LIN {X 0,Y 154.831,Z 493.281,A -85,B 0,C 180,E1 -25779.499,E2 -25779.499} C_VEL
LIN {X 0,Y 149.043,Z 503.772,A -85,B 0,C 180,E1 -25782.041,E2 -25782.041} C_VEL
LIN {X 0,Y 142.344,Z 514.195,A -85,B 0,C 180,E1 -25785.287,E2 -25785.287} C_VEL
LIN {X 0,Y 136.226,Z 522.789,A -85,B 0,C 180,E1 -25788.87,E2 -25788.87} C_VEL
LIN {X 0,Y 129.735,Z 531.025,A -85,B 0,C 180,E1 -25793.425,E2 -25793.425} C_VEL
LIN {X 0,Y 124.804,Z 536.98,A -85,B 0,C 180,E1 -25797.884,E2 -25797.884} C_VEL
LIN {X 0,Y 119.794,Z 542.879,A -85,B 0,C 180,E1 -25803.896,E2 -25803.896} C_VEL
LIN {X 0,Y 116.608,Z 546.367,A -85,B 0,C 180,E1 -25808.8,E2 -25808.8} C_VEL
LIN {X 0,Y 113.843,Z 549.761,A -85,B 0,C 180,E1 -25815.704,E2 -25815.704} C_VEL
LIN {X 0,Y 112.436,Z 551.771,A -85,B 0,C 180,E1 -25822.818,E2 -25822.818} C_VEL
LIN {X 0,Y 112.199,Z 552.451,A -85,B 0,C 180,E1 -25830,E2 -25830} C_VEL
LIN {X 0,Y 112.434,Z 551.816,A -85,B 0,C 180,E1 -25837.181,E2 -25837.181} C_VEL
LIN {X 0,Y 113.819,Z 549.846,A -85,B 0,C 180,E1 -25844.299,E2 -25844.299} C_VEL
LIN {X 0,Y 116.58,Z 546.493,A -85,B 0,C 180,E1 -25851.204,E2 -25851.204} C_VEL
LIN {X 0,Y 120.927,Z 541.656,A -85,B 0,C 180,E1 -25857.706,E2 -25857.706} C_VEL
LIN {X 0,Y 126.423,Z 535.183,A -85,B 0,C 180,E1 -25863.773,E2 -25863.773} C_VEL
LIN {X 0,Y 132.35,Z 527.972,A -85,B 0,C 180,E1 -25868.603,E2 -25868.603} C_VEL
LIN {X 0,Y 139.146,Z 519.048,A -85,B 0,C 180,E1 -25872.988,E2 -25872.988} C_VEL
LIN {X 0,Y 145.538,Z 509.671,A -85,B 0,C 180,E1 -25876.413,E2 -25876.413} C_VEL
LIN {X 0,Y 151.745,Z 499.424,A -85,B 0,C 180,E1 -25879.256,E2 -25879.256} C_VEL
LIN {X 0,Y 157.702,Z 487.826,A -85,B 0,C 180,E1 -25881.761,E2 -25881.761} C_VEL
LIN {X 0,Y 163.296,Z 475.115,A -85,B 0,C 180,E1 -25883.799,E2 -25883.799} C_VEL
LIN {X 0,Y 167.805,Z 462.736,A -85,B 0,C 180,E1 -25885.277,E2 -25885.277} C_VEL
LIN {X 0,Y 171.372,Z 450.293,A -85,B 0,C 180,E1 -25886.408,E2 -25886.408} C_VEL
LIN {X 0,Y 174.368,Z 436.456,A -85,B 0,C 180,E1 -25887.284,E2 -25887.284} C_VEL
LIN {X 0,Y 176.327,Z 422.007,A -85,B 0,C 180,E1 -25887.898,E2 -25887.898} C_VEL
LIN {X 0,Y 179.543,Z 385.834,A -85,B 0,C 180,E1 -25888.964,E2 -25888.964} C_VEL
LIN {X 0,Y 177.542,Z 380.775,A -85,B 0,C 180,E1 -25890.461,E2 -25890.461} C_VEL
LIN {X 0,Y 173.513,Z 372.831,A -85,B 0,C 180,E1 -25893.622,E2 -25893.622} C_VEL
LIN {X 0,Y 169.768,Z 366.134,A -85,B 0,C 180,E1 -25897.004,E2 -25897.004} C_VEL
LIN {X 0,Y 166.328,Z 360.29,A -85,B 0,C 180,E1 -25900.724,E2 -25900.724} C_VEL
LIN {X 0,Y 163.415,Z 355.804,A -85,B 0,C 180,E1 -25904.621,E2 -25904.621} C_VEL
LIN {X 0,Y 161.232,Z 352.232,A -85,B 0,C 180,E1 -25908.528,E2 -25908.528} C_VEL
LIN {X 0,Y 158.664,Z 347.179,A -85,B 0,C 180,E1 -25919.365,E2 -25919.365} C_VEL
LIN {X 0,Y 158.668,Z 347.413,A -85,B 0,C 180,E1 -25921.269,E2 -25921.269} C_VEL
LIN {X 0,Y 161.202,Z 352.144,A -85,B 0,C 180,E1 -25931.314,E2 -25931.314} C_VEL
LIN {X 0,Y 163.612,Z 356.049,A -85,B 0,C 180,E1 -25935.581,E2 -25935.581} C_VEL
LIN {X 0,Y 166.843,Z 361.285,A -85,B 0,C 180,E1 -25939.813,E2 -25939.813} C_VEL
LIN {X 0,Y 169.27,Z 365.259,A -85,B 0,C 180,E1 -25942.412,E2 -25942.412} C_VEL
LIN {X 0,Y 172.886,Z 371.75,A -85,B 0,C 180,E1 -25945.767,E2 -25945.767} C_VEL
LIN {X 0,Y 174.889,Z 375.758,A -85,B 0,C 180,E1 -25947.444,E2 -25947.444} C_VEL
LIN {X 0,Y 177.962,Z 383.47,A -85,B 0,C 180,E1 -25949.905,E2 -25949.905} C_VEL
LIN {X 0,Y 179.384,Z 387.559,A -85,B 0,C 180,E1 -25950.996,E2 -25950.996} C_VEL
LIN {X 0,Y 175.579,Z 429.688,A -85,B 0,C 180,E1 -25952.309,E2 -25952.309} C_VEL
LIN {X 0,Y 173.1,Z 443.982,A -85,B 0,C 180,E1 -25953.004,E2 -25953.004} C_VEL
LIN {X 0,Y 169.543,Z 457.949,A -85,B 0,C 180,E1 -25954.001,E2 -25954.001} C_VEL
LIN {X 0,Y 164.994,Z 471.812,A -85,B 0,C 180,E1 -25955.45,E2 -25955.45} C_VEL
LIN {X 0,Y 159.867,Z 484.227,A -85,B 0,C 180,E1 -25957.176,E2 -25957.176} C_VEL
LIN {X 0,Y 154.341,Z 495.58,A -85,B 0,C 180,E1 -25959.278,E2 -25959.278} C_VEL
LIN {X 0,Y 148.493,Z 506.017,A -85,B 0,C 180,E1 -25961.806,E2 -25961.806} C_VEL
LIN {X 0,Y 141.881,Z 516.403,A -85,B 0,C 180,E1 -25965.102,E2 -25965.102} C_VEL
LIN {X 0,Y 135.687,Z 524.971,A -85,B 0,C 180,E1 -25968.671,E2 -25968.671} C_VEL
LIN {X 0,Y 129.237,Z 533.17,A -85,B 0,C 180,E1 -25973.261,E2 -25973.261} C_VEL
LIN {X 0,Y 123.346,Z 540.219,A -85,B 0,C 180,E1 -25978.723,E2 -25978.723} C_VEL
LIN {X 0,Y 119.298,Z 545.014,A -85,B 0,C 180,E1 -25983.78,E2 -25983.78} C_VEL
LIN {X 0,Y 116.235,Z 548.502,A -85,B 0,C 180,E1 -25988.73,E2 -25988.73} C_VEL
LIN {X 0,Y 113.556,Z 551.894,A -85,B 0,C 180,E1 -25995.667,E2 -25995.667} C_VEL
LIN {X 0,Y 112.263,Z 553.898,A -85,B 0,C 180,E1 -26002.808,E2 -26002.808} C_VEL
LIN {X 0,Y 112.133,Z 554.556,A -85,B 0,C 180,E1 -26010,E2 -26010} C_VEL
LIN {X 0,Y 112.278,Z 553.828,A -85,B 0,C 180,E1 -26017.38,E2 -26017.38} C_VEL
LIN {X 0,Y 113.582,Z 551.845,A -85,B 0,C 180,E1 -26024.33,E2 -26024.33} C_VEL
LIN {X 0,Y 116.237,Z 548.428,A -85,B 0,C 180,E1 -26031.271,E2 -26031.271} C_VEL
LIN {X 0,Y 116.783,Z 547.806,A -85,B 0,C 180,E1 -26032.245,E2 -26032.245} C_VEL
LIN {X 0,Y 117.755,Z 546.031,A -85,B 0,C 180,E1 -26034.955,E2 -26034.955} C_VEL
LIN {X 0,Y 118.012,Z 542.788,A -85,B 0,C 180,E1 -26039.51,E2 -26039.51} C_VEL
LIN {X 0,Y 118.831,Z 538.965,A -85,B 0,C 180,E1 -26043.93,E2 -26043.93} C_VEL
LIN {X 0,Y 120.612,Z 536.281,A -85,B 0,C 180,E1 -26046.303,E2 -26046.303} C_VEL
LIN {X 0,Y 126.397,Z 529.621,A -85,B 0,C 180,E1 -26050.792,E2 -26050.792} C_VEL
LIN {X 0,Y 133.529,Z 520.595,A -85,B 0,C 180,E1 -26055.278,E2 -26055.278} C_VEL
LIN {X 0,Y 140.331,Z 511.13,A -85,B 0,C 180,E1 -26058.695,E2 -26058.695} C_VEL
LIN {X 0,Y 146.494,Z 501.341,A -85,B 0,C 180,E1 -26061.416,E2 -26061.416} C_VEL
LIN {X 0,Y 152.443,Z 490.369,A -85,B 0,C 180,E1 -26063.782,E2 -26063.782} C_VEL
LIN {X 0,Y 158.317,Z 477.817,A -85,B 0,C 180,E1 -26065.77,E2 -26065.77} C_VEL
LIN {X 0,Y 162.993,Z 465.66,A -85,B 0,C 180,E1 -26067.224,E2 -26067.224} C_VEL
LIN {X 0,Y 167.084,Z 452.297,A -85,B 0,C 180,E1 -26068.396,E2 -26068.396} C_VEL
LIN {X 0,Y 170.16,Z 438.671,A -85,B 0,C 180,E1 -26069.249,E2 -26069.249} C_VEL
LIN {X 0,Y 172.249,Z 424.594,A -85,B 0,C 180,E1 -26069.814,E2 -26069.814} C_VEL
LIN {X 0,Y 175.377,Z 390.18,A -85,B 0,C 180,E1 -26070.85,E2 -26070.85} C_VEL
LIN {X 0,Y 172.372,Z 381.864,A -85,B 0,C 180,E1 -26073.435,E2 -26073.435} C_VEL
LIN {X 0,Y 170.665,Z 378.041,A -85,B 0,C 180,E1 -26074.969,E2 -26074.969} C_VEL
LIN {X 0,Y 167.157,Z 371.404,A -85,B 0,C 180,E1 -26078.415,E2 -26078.415} C_VEL
LIN {X 0,Y 164.04,Z 366.093,A -85,B 0,C 180,E1 -26082.065,E2 -26082.065} C_VEL
LIN {X 0,Y 161.76,Z 362.326,A -85,B 0,C 180,E1 -26085.373,E2 -26085.373} C_VEL
LIN {X 0,Y 159.691,Z 358.606,A -85,B 0,C 180,E1 -26089.38,E2 -26089.38} C_VEL
LIN {X 0,Y 157.511,Z 354.085,A -85,B 0,C 180,E1 -26098.722,E2 -26098.722} C_VEL
LIN {X 0,Y 157.506,Z 354.034,A -85,B 0,C 180,E1 -26101.279,E2 -26101.279} C_VEL
LIN {X 0,Y 159.956,Z 359.128,A -85,B 0,C 180,E1 -26111.404,E2 -26111.404} C_VEL
LIN {X 0,Y 162.479,Z 363.489,A -85,B 0,C 180,E1 -26115.926,E2 -26115.926} C_VEL
LIN {X 0,Y 164.967,Z 367.653,A -85,B 0,C 180,E1 -26119.279,E2 -26119.279} C_VEL
LIN {X 0,Y 167.552,Z 372.121,A -85,B 0,C 180,E1 -26122.18,E2 -26122.18} C_VEL
LIN {X 0,Y 171.277,Z 379.139,A -85,B 0,C 180,E1 -26125.746,E2 -26125.746} C_VEL
LIN {X 0,Y 175.153,Z 387.363,A -85,B 0,C 180,E1 -26128.962,E2 -26128.962} C_VEL
LIN {X 0,Y 175.509,Z 388.434,A -85,B 0,C 180,E1 -26129.26,E2 -26129.26} C_VEL
LIN {X 0,Y 171.755,Z 428.026,A -85,B 0,C 180,E1 -26130.46,E2 -26130.46} C_VEL
LIN {X 0,Y 169.296,Z 442.095,A -85,B 0,C 180,E1 -26131.155,E2 -26131.155} C_VEL
LIN {X 0,Y 165.594,Z 456.476,A -85,B 0,C 180,E1 -26132.204,E2 -26132.204} C_VEL
LIN {X 0,Y 161.246,Z 469.396,A -85,B 0,C 180,E1 -26133.534,E2 -26133.534} C_VEL
LIN {X 0,Y 156.036,Z 481.927,A -85,B 0,C 180,E1 -26135.279,E2 -26135.279} C_VEL
LIN {X 0,Y 150.311,Z 493.509,A -85,B 0,C 180,E1 -26137.433,E2 -26137.433} C_VEL
LIN {X 0,Y 144.379,Z 503.842,A -85,B 0,C 180,E1 -26139.946,E2 -26139.946} C_VEL
LIN {X 0,Y 137.381,Z 514.264,A -85,B 0,C 180,E1 -26143.199,E2 -26143.199} C_VEL
LIN {X 0,Y 130.954,Z 522.858,A -85,B 0,C 180,E1 -26146.823,E2 -26146.823} C_VEL
LIN {X 0,Y 124.087,Z 531.093,A -85,B 0,C 180,E1 -26151.464,E2 -26151.464} C_VEL
LIN {X 0,Y 119.119,Z 536.642,A -85,B 0,C 180,E1 -26155.691,E2 -26155.691} C_VEL
LIN {X 0,Y 114.718,Z 541.549,A -85,B 0,C 180,E1 -26160.653,E2 -26160.653} C_VEL
LIN {X 0,Y 109.986,Z 546.435,A -85,B 0,C 180,E1 -26167.456,E2 -26167.456} C_VEL
LIN {X 0,Y 106.95,Z 549.829,A -85,B 0,C 180,E1 -26174.761,E2 -26174.761} C_VEL
LIN {X 0,Y 105.378,Z 551.838,A -85,B 0,C 180,E1 -26182.335,E2 -26182.335} C_VEL
LIN {X 0,Y 105.106,Z 552.518,A -85,B 0,C 180,E1 -26190,E2 -26190} C_VEL
LIN {X 0,Y 105.373,Z 551.883,A -85,B 0,C 180,E1 -26197.665,E2 -26197.665} C_VEL
LIN {X 0,Y 106.929,Z 549.912,A -85,B 0,C 180,E1 -26205.242,E2 -26205.242} C_VEL
LIN {X 0,Y 109.96,Z 546.559,A -85,B 0,C 180,E1 -26212.549,E2 -26212.549} C_VEL
LIN {X 0,Y 114.642,Z 541.722,A -85,B 0,C 180,E1 -26219.368,E2 -26219.368} C_VEL
LIN {X 0,Y 120.56,Z 535.248,A -85,B 0,C 180,E1 -26225.657,E2 -26225.657} C_VEL
LIN {X 0,Y 126.86,Z 528.037,A -85,B 0,C 180,E1 -26230.612,E2 -26230.612} C_VEL
LIN {X 0,Y 134.008,Z 519.113,A -85,B 0,C 180,E1 -26235.071,E2 -26235.071} C_VEL
LIN {X 0,Y 140.732,Z 509.734,A -85,B 0,C 180,E1 -26238.509,E2 -26238.509} C_VEL
LIN {X 0,Y 146.984,Z 499.861,A -85,B 0,C 180,E1 -26241.268,E2 -26241.268} C_VEL
LIN {X 0,Y 153.404,Z 487.888,A -85,B 0,C 180,E1 -26243.847,E2 -26243.847} C_VEL
LIN {X 0,Y 159.21,Z 475.176,A -85,B 0,C 180,E1 -26245.859,E2 -26245.859} C_VEL
LIN {X 0,Y 163.865,Z 462.797,A -85,B 0,C 180,E1 -26247.317,E2 -26247.317} C_VEL
LIN {X 0,Y 167.556,Z 450.351,A -85,B 0,C 180,E1 -26248.427,E2 -26248.427} C_VEL
LIN {X 0,Y 170.642,Z 436.511,A -85,B 0,C 180,E1 -26249.286,E2 -26249.286} C_VEL
LIN {X 0,Y 172.672,Z 422.053,A -85,B 0,C 180,E1 -26249.887,E2 -26249.887} C_VEL
LIN {X 0,Y 175.751,Z 388.718,A -85,B 0,C 180,E1 -26250.849,E2 -26250.849} C_VEL
LIN {X 0,Y 173.862,Z 384.198,A -85,B 0,C 180,E1 -26252.38,E2 -26252.38} C_VEL
LIN {X 0,Y 169.806,Z 376.049,A -85,B 0,C 180,E1 -26255.944,E2 -26255.944} C_VEL
LIN {X 0,Y 166.416,Z 369.87,A -85,B 0,C 180,E1 -26259.448,E2 -26259.448} C_VEL
LIN {X 0,Y 164.261,Z 366.273,A -85,B 0,C 180,E1 -26262.058,E2 -26262.058} C_VEL
LIN {X 0,Y 161.985,Z 362.452,A -85,B 0,C 180,E1 -26265.393,E2 -26265.393} C_VEL
LIN {X 0,Y 159.727,Z 358.589,A -85,B 0,C 180,E1 -26269.863,E2 -26269.863} C_VEL
LIN {X 0,Y 157.802,Z 354.129,A -85,B 0,C 180,E1 -26280,E2 -26280} C_VEL
LIN {X 0,Y 160.021,Z 358.971,A -85,B 0,C 180,E1 -26290.718,E2 -26290.718} C_VEL
LIN {X 0,Y 162.659,Z 363.601,A -85,B 0,C 180,E1 -26295.593,E2 -26295.593} C_VEL
LIN {X 0,Y 165.295,Z 368.002,A -85,B 0,C 180,E1 -26299.159,E2 -26299.159} C_VEL
LIN {X 0,Y 168.289,Z 373.184,A -85,B 0,C 180,E1 -26302.471,E2 -26302.471} C_VEL
LIN {X 0,Y 171.793,Z 380.078,A -85,B 0,C 180,E1 -26305.797,E2 -26305.797} C_VEL
LIN {X 0,Y 174.641,Z 387.517,A -85,B 0,C 180,E1 -26308.301,E2 -26308.301} C_VEL
LIN {X 0,Y 175.601,Z 390.329,A -85,B 0,C 180,E1 -26309.109,E2 -26309.109} C_VEL
LIN {X 0,Y 171.889,Z 429.635,A -85,B 0,C 180,E1 -26310.308,E2 -26310.308} C_VEL
LIN {X 0,Y 169.343,Z 443.925,A -85,B 0,C 180,E1 -26310.991,E2 -26310.991} C_VEL
LIN {X 0,Y 165.677,Z 457.89,A -85,B 0,C 180,E1 -26311.965,E2 -26311.965} C_VEL
LIN {X 0,Y 160.969,Z 471.751,A -85,B 0,C 180,E1 -26313.385,E2 -26313.385} C_VEL
LIN {X 0,Y 155.67,Z 484.165,A -85,B 0,C 180,E1 -26315.089,E2 -26315.089} C_VEL
LIN {X 0,Y 149.929,Z 495.517,A -85,B 0,C 180,E1 -26317.168,E2 -26317.168} C_VEL
LIN {X 0,Y 143.85,Z 505.953,A -85,B 0,C 180,E1 -26319.694,E2 -26319.694} C_VEL
LIN {X 0,Y 136.928,Z 516.338,A -85,B 0,C 180,E1 -26322.998,E2 -26322.998} C_VEL
LIN {X 0,Y 130.406,Z 524.906,A -85,B 0,C 180,E1 -26326.598,E2 -26326.598} C_VEL
LIN {X 0,Y 123.579,Z 533.104,A -85,B 0,C 180,E1 -26331.277,E2 -26331.277} C_VEL
LIN {X 0,Y 118.498,Z 538.854,A -85,B 0,C 180,E1 -26335.707,E2 -26335.707} C_VEL
LIN {X 0,Y 114.217,Z 543.56,A -85,B 0,C 180,E1 -26340.512,E2 -26340.512} C_VEL
LIN {X 0,Y 109.632,Z 548.437,A -85,B 0,C 180,E1 -26347.38,E2 -26347.38} C_VEL
LIN {X 0,Y 106.642,Z 551.828,A -85,B 0,C 180,E1 -26354.716,E2 -26354.716} C_VEL
LIN {X 0,Y 105.221,Z 553.832,A -85,B 0,C 180,E1 -26362.324,E2 -26362.324} C_VEL
LIN {X 0,Y 105.033,Z 554.489,A -85,B 0,C 180,E1 -26370,E2 -26370} C_VEL
LIN {X 0,Y 105.222,Z 553.805,A -85,B 0,C 180,E1 -26377.677,E2 -26377.677} C_VEL
LIN {X 0,Y 106.665,Z 551.778,A -85,B 0,C 180,E1 -26385.281,E2 -26385.281} C_VEL
LIN {X 0,Y 109.633,Z 548.36,A -85,B 0,C 180,E1 -26392.62,E2 -26392.62} C_VEL
LIN {X 0,Y 114.167,Z 543.45,A -85,B 0,C 180,E1 -26399.503,E2 -26399.503} C_VEL
LIN {X 0,Y 118.45,Z 538.716,A -85,B 0,C 180,E1 -26404.309,E2 -26404.309} C_VEL
LIN {X 0,Y 120.612,Z 536.281,A -85,B 0,C 180,E1 -26406.303,E2 -26406.303} C_VEL
LIN {X 0,Y 122.566,Z 533.459,A -85,B 0,C 180,E1 -26408.571,E2 -26408.571} C_VEL
LIN {X 0,Y 124.537,Z 528.588,A -85,B 0,C 180,E1 -26412.492,E2 -26412.492} C_VEL
LIN {X 0,Y 126.904,Z 523.234,A -85,B 0,C 180,E1 -26416.137,E2 -26416.137} C_VEL
LIN {X 0,Y 129.353,Z 519.595,A -85,B 0,C 180,E1 -26417.9,E2 -26417.9} C_VEL
LIN {X 0,Y 136.961,Z 509.277,A -85,B 0,C 180,E1 -26421.492,E2 -26421.492} C_VEL
LIN {X 0,Y 143.63,Z 498.759,A -85,B 0,C 180,E1 -26424.256,E2 -26424.256} C_VEL
LIN {X 0,Y 149.688,Z 487.715,A -85,B 0,C 180,E1 -26426.446,E2 -26426.446} C_VEL
LIN {X 0,Y 155.114,Z 476.163,A -85,B 0,C 180,E1 -26428.159,E2 -26428.159} C_VEL
LIN {X 0,Y 160.305,Z 462.603,A -85,B 0,C 180,E1 -26429.668,E2 -26429.668} C_VEL
LIN {X 0,Y 164.387,Z 448.805,A -85,B 0,C 180,E1 -26430.769,E2 -26430.769} C_VEL
LIN {X 0,Y 167.429,Z 434.454,A -85,B 0,C 180,E1 -26431.527,E2 -26431.527} C_VEL
LIN {X 0,Y 169.386,Z 418.688,A -85,B 0,C 180,E1 -26432.07,E2 -26432.07} C_VEL
LIN {X 0,Y 171.756,Z 393.082,A -85,B 0,C 180,E1 -26432.826,E2 -26432.826} C_VEL
LIN {X 0,Y 169.09,Z 385.396,A -85,B 0,C 180,E1 -26435.389,E2 -26435.389} C_VEL
LIN {X 0,Y 165.703,Z 378.484,A -85,B 0,C 180,E1 -26438.87,E2 -26438.87} C_VEL
LIN {X 0,Y 162.588,Z 372.799,A -85,B 0,C 180,E1 -26442.712,E2 -26442.712} C_VEL
LIN {X 0,Y 160.329,Z 368.884,A -85,B 0,C 180,E1 -26446.211,E2 -26446.211} C_VEL
LIN {X 0,Y 158.475,Z 365.407,A -85,B 0,C 180,E1 -26450.105,E2 -26450.105} C_VEL
LIN {X 0,Y 156.641,Z 361.17,A -85,B 0,C 180,E1 -26458.715,E2 -26458.715} C_VEL
LIN {X 0,Y 156.625,Z 360.935,A -85,B 0,C 180,E1 -26460,E2 -26460} C_VEL
LIN {X 0,Y 156.664,Z 361.526,A -85,B 0,C 180,E1 -26462.25,E2 -26462.25} C_VEL
LIN {X 0,Y 158.792,Z 365.998,A -85,B 0,C 180,E1 -26470.842,E2 -26470.842} C_VEL
LIN {X 0,Y 161.048,Z 370.137,A -85,B 0,C 180,E1 -26475.179,E2 -26475.179} C_VEL
LIN {X 0,Y 163.413,Z 374.316,A -85,B 0,C 180,E1 -26478.574,E2 -26478.574} C_VEL
LIN {X 0,Y 166.258,Z 379.525,A -85,B 0,C 180,E1 -26481.913,E2 -26481.913} C_VEL
LIN {X 0,Y 170.019,Z 387.29,A -85,B 0,C 180,E1 -26485.642,E2 -26485.642} C_VEL
LIN {X 0,Y 171.891,Z 391.502,A -85,B 0,C 180,E1 -26487.297,E2 -26487.297} C_VEL
LIN {X 0,Y 168.155,Z 428.91,A -85,B 0,C 180,E1 -26488.416,E2 -26488.416} C_VEL
LIN {X 0,Y 165.533,Z 443.044,A -85,B 0,C 180,E1 -26489.109,E2 -26489.109} C_VEL
LIN {X 0,Y 161.927,Z 456.55,A -85,B 0,C 180,E1 -26490.081,E2 -26490.081} C_VEL
LIN {X 0,Y 157.437,Z 469.468,A -85,B 0,C 180,E1 -26491.381,E2 -26491.381} C_VEL
LIN {X 0,Y 152.04,Z 481.998,A -85,B 0,C 180,E1 -26493.091,E2 -26493.091} C_VEL
LIN {X 0,Y 146.165,Z 493.423,A -85,B 0,C 180,E1 -26495.175,E2 -26495.175} C_VEL
LIN {X 0,Y 139.922,Z 503.912,A -85,B 0,C 180,E1 -26497.714,E2 -26497.714} C_VEL
LIN {X 0,Y 132.615,Z 514.334,A -85,B 0,C 180,E1 -26500.96,E2 -26500.96} C_VEL
LIN {X 0,Y 125.852,Z 522.927,A -85,B 0,C 180,E1 -26504.603,E2 -26504.603} C_VEL
LIN {X 0,Y 118.592,Z 531.162,A -85,B 0,C 180,E1 -26509.317,E2 -26509.317} C_VEL
LIN {X 0,Y 112.947,Z 537.089,A -85,B 0,C 180,E1 -26513.99,E2 -26513.99} C_VEL
LIN {X 0,Y 107.177,Z 543.015,A -85,B 0,C 180,E1 -26520.541,E2 -26520.541} C_VEL
LIN {X 0,Y 103.436,Z 546.502,A -85,B 0,C 180,E1 -26525.942,E2 -26525.942} C_VEL
LIN {X 0,Y 100.098,Z 549.896,A -85,B 0,C 180,E1 -26533.69,E2 -26533.69} C_VEL
LIN {X 0,Y 98.336,Z 551.905,A -85,B 0,C 180,E1 -26541.782,E2 -26541.782} C_VEL
LIN {X 0,Y 98.006,Z 552.585,A -85,B 0,C 180,E1 -26550,E2 -26550} C_VEL
LIN {X 0,Y 98.33,Z 551.949,A -85,B 0,C 180,E1 -26558.218,E2 -26558.218} C_VEL
LIN {X 0,Y 100.079,Z 549.978,A -85,B 0,C 180,E1 -26566.313,E2 -26566.313} C_VEL
LIN {X 0,Y 103.412,Z 546.625,A -85,B 0,C 180,E1 -26574.064,E2 -26574.064} C_VEL
LIN {X 0,Y 108.469,Z 541.788,A -85,B 0,C 180,E1 -26581.22,E2 -26581.22} C_VEL
LIN {X 0,Y 114.826,Z 535.314,A -85,B 0,C 180,E1 -26587.737,E2 -26587.737} C_VEL
LIN {X 0,Y 121.548,Z 528.102,A -85,B 0,C 180,E1 -26592.795,E2 -26592.795} C_VEL
LIN {X 0,Y 129.068,Z 519.177,A -85,B 0,C 180,E1 -26597.314,E2 -26597.314} C_VEL
LIN {X 0,Y 136.124,Z 509.798,A -85,B 0,C 180,E1 -26600.753,E2 -26600.753} C_VEL
LIN {X 0,Y 143.307,Z 498.715,A -85,B 0,C 180,E1 -26603.808,E2 -26603.808} C_VEL
LIN {X 0,Y 149.972,Z 486.66,A -85,B 0,C 180,E1 -26606.282,E2 -26606.282} C_VEL
LIN {X 0,Y 155.337,Z 475.238,A -85,B 0,C 180,E1 -26608.027,E2 -26608.027} C_VEL
LIN {X 0,Y 160.139,Z 462.857,A -85,B 0,C 180,E1 -26609.458,E2 -26609.458} C_VEL
LIN {X 0,Y 164.264,Z 449.283,A -85,B 0,C 180,E1 -26610.617,E2 -26610.617} C_VEL
LIN {X 0,Y 167.359,Z 435.332,A -85,B 0,C 180,E1 -26611.445,E2 -26611.445} C_VEL
LIN {X 0,Y 169.329,Z 421.189,A -85,B 0,C 180,E1 -26611.994,E2 -26611.994} C_VEL
LIN {X 0,Y 172.133,Z 391.736,A -85,B 0,C 180,E1 -26612.82,E2 -26612.82} C_VEL
LIN {X 0,Y 168.615,Z 384.111,A -85,B 0,C 180,E1 -26616.027,E2 -26616.027} C_VEL
LIN {X 0,Y 165.63,Z 378.137,A -85,B 0,C 180,E1 -26619.176,E2 -26619.176} C_VEL
LIN {X 0,Y 162.68,Z 372.786,A -85,B 0,C 180,E1 -26622.884,E2 -26622.884} C_VEL
LIN {X 0,Y 160.554,Z 369.057,A -85,B 0,C 180,E1 -26626.23,E2 -26626.23} C_VEL
LIN {X 0,Y 158.66,Z 365.533,A -85,B 0,C 180,E1 -26630.277,E2 -26630.277} C_VEL
LIN {X 0,Y 156.934,Z 361.2,A -85,B 0,C 180,E1 -26640,E2 -26640} C_VEL
LIN {X 0,Y 158.886,Z 365.886,A -85,B 0,C 180,E1 -26650.191,E2 -26650.191} C_VEL
LIN {X 0,Y 161.185,Z 370.158,A -85,B 0,C 180,E1 -26654.762,E2 -26654.762} C_VEL
LIN {X 0,Y 163.654,Z 374.504,A -85,B 0,C 180,E1 -26658.343,E2 -26658.343} C_VEL
LIN {X 0,Y 166.29,Z 379.356,A -85,B 0,C 180,E1 -26661.47,E2 -26661.47} C_VEL
LIN {X 0,Y 169.511,Z 386.132,A -85,B 0,C 180,E1 -26664.761,E2 -26664.761} C_VEL
LIN {X 0,Y 171.977,Z 393.158,A -85,B 0,C 180,E1 -26667.12,E2 -26667.12} C_VEL
LIN {X 0,Y 168.347,Z 430.051,A -85,B 0,C 180,E1 -26668.242,E2 -26668.242} C_VEL
LIN {X 0,Y 165.723,Z 444.22,A -85,B 0,C 180,E1 -26668.912,E2 -26668.912} C_VEL
LIN {X 0,Y 162.031,Z 457.83,A -85,B 0,C 180,E1 -26669.834,E2 -26669.834} C_VEL
LIN {X 0,Y 157.161,Z 471.689,A -85,B 0,C 180,E1 -26671.216,E2 -26671.216} C_VEL
LIN {X 0,Y 151.698,Z 484.102,A -85,B 0,C 180,E1 -26672.893,E2 -26672.893} C_VEL
LIN {X 0,Y 145.734,Z 495.453,A -85,B 0,C 180,E1 -26674.935,E2 -26674.935} C_VEL
LIN {X 0,Y 139.42,Z 505.89,A -85,B 0,C 180,E1 -26677.447,E2 -26677.447} C_VEL
LIN {X 0,Y 132.167,Z 516.274,A -85,B 0,C 180,E1 -26680.736,E2 -26680.736} C_VEL
LIN {X 0,Y 125.318,Z 524.841,A -85,B 0,C 180,E1 -26684.355,E2 -26684.355} C_VEL
LIN {X 0,Y 118.101,Z 533.039,A -85,B 0,C 180,E1 -26689.113,E2 -26689.113} C_VEL
LIN {X 0,Y 112.653,Z 538.789,A -85,B 0,C 180,E1 -26693.654,E2 -26693.654} C_VEL
LIN {X 0,Y 106.658,Z 544.882,A -85,B 0,C 180,E1 -26700.384,E2 -26700.384} C_VEL
LIN {X 0,Y 103.097,Z 548.371,A -85,B 0,C 180,E1 -26705.858,E2 -26705.858} C_VEL
LIN {X 0,Y 99.769,Z 551.761,A -85,B 0,C 180,E1 -26713.635,E2 -26713.635} C_VEL
LIN {X 0,Y 98.178,Z 553.765,A -85,B 0,C 180,E1 -26721.769,E2 -26721.769} C_VEL
LIN {X 0,Y 97.94,Z 554.423,A -85,B 0,C 180,E1 -26730,E2 -26730} C_VEL
LIN {X 0,Y 98.179,Z 553.738,A -85,B 0,C 180,E1 -26738.231,E2 -26738.231} C_VEL
LIN {X 0,Y 99.787,Z 551.71,A -85,B 0,C 180,E1 -26746.363,E2 -26746.363} C_VEL
LIN {X 0,Y 103.097,Z 548.293,A -85,B 0,C 180,E1 -26754.143,E2 -26754.143} C_VEL
LIN {X 0,Y 107.998,Z 543.382,A -85,B 0,C 180,E1 -26761.372,E2 -26761.372} C_VEL
LIN {X 0,Y 112.625,Z 538.647,A -85,B 0,C 180,E1 -26766.356,E2 -26766.356} C_VEL
LIN {X 0,Y 119.061,Z 531.788,A -85,B 0,C 180,E1 -26771.61,E2 -26771.61} C_VEL
LIN {X 0,Y 126.365,Z 523.274,A -85,B 0,C 180,E1 -26776.303,E2 -26776.303} C_VEL
LIN {X 0,Y 129.353,Z 519.595,A -85,B 0,C 180,E1 -26777.9,E2 -26777.9} C_VEL
LIN {X 0,Y 131.849,Z 515.843,A -85,B 0,C 180,E1 -26779.549,E2 -26779.549} C_VEL
LIN {X 0,Y 134.662,Z 509.463,A -85,B 0,C 180,E1 -26782.587,E2 -26782.587} C_VEL
LIN {X 0,Y 137.474,Z 502.736,A -85,B 0,C 180,E1 -26785.425,E2 -26785.425} C_VEL
LIN {X 0,Y 139.848,Z 498.27,A -85,B 0,C 180,E1 -26786.724,E2 -26786.724} C_VEL
LIN {X 0,Y 145.882,Z 487.644,A -85,B 0,C 180,E1 -26788.772,E2 -26788.772} C_VEL
LIN {X 0,Y 151.492,Z 476.091,A -85,B 0,C 180,E1 -26790.439,E2 -26790.439} C_VEL
LIN {X 0,Y 156.846,Z 462.53,A -85,B 0,C 180,E1 -26791.902,E2 -26791.902} C_VEL
LIN {X 0,Y 160.898,Z 449.259,A -85,B 0,C 180,E1 -26792.936,E2 -26792.936} C_VEL
LIN {X 0,Y 164.048,Z 435.053,A -85,B 0,C 180,E1 -26793.684,E2 -26793.684} C_VEL
LIN {X 0,Y 166.152,Z 418.942,A -85,B 0,C 180,E1 -26794.219,E2 -26794.219} C_VEL
LIN {X 0,Y 168.328,Z 395.923,A -85,B 0,C 180,E1 -26794.905,E2 -26794.905} C_VEL
LIN {X 0,Y 166.227,Z 389.923,A -85,B 0,C 180,E1 -26797.135,E2 -26797.135} C_VEL
LIN {X 0,Y 163.037,Z 383.162,A -85,B 0,C 180,E1 -26800.811,E2 -26800.811} C_VEL
LIN {X 0,Y 160.716,Z 378.768,A -85,B 0,C 180,E1 -26804.017,E2 -26804.017} C_VEL
LIN {X 0,Y 158.846,Z 375.34,A -85,B 0,C 180,E1 -26807.219,E2 -26807.219} C_VEL
LIN {X 0,Y 157.351,Z 372.252,A -85,B 0,C 180,E1 -26810.682,E2 -26810.682} C_VEL
LIN {X 0,Y 155.76,Z 368.083,A -85,B 0,C 180,E1 -26819.354,E2 -26819.354} C_VEL
LIN {X 0,Y 155.768,Z 368.36,A -85,B 0,C 180,E1 -26821.616,E2 -26821.616} C_VEL
LIN {X 0,Y 157.603,Z 372.722,A -85,B 0,C 180,E1 -26830.154,E2 -26830.154} C_VEL
LIN {X 0,Y 159.746,Z 376.961,A -85,B 0,C 180,E1 -26834.589,E2 -26834.589} C_VEL
LIN {X 0,Y 161.937,Z 381.105,A -85,B 0,C 180,E1 -26837.931,E2 -26837.931} C_VEL
LIN {X 0,Y 164.564,Z 386.261,A -85,B 0,C 180,E1 -26841.203,E2 -26841.203} C_VEL
LIN {X 0,Y 167.667,Z 393.111,A -85,B 0,C 180,E1 -26844.503,E2 -26844.503} C_VEL
LIN {X 0,Y 168.423,Z 394.879,A -85,B 0,C 180,E1 -26845.238,E2 -26845.238} C_VEL
LIN {X 0,Y 164.912,Z 428.876,A -85,B 0,C 180,E1 -26846.24,E2 -26846.24} C_VEL
LIN {X 0,Y 162.137,Z 443.368,A -85,B 0,C 180,E1 -26846.93,E2 -26846.93} C_VEL
LIN {X 0,Y 158.127,Z 457.753,A -85,B 0,C 180,E1 -26847.953,E2 -26847.953} C_VEL
LIN {X 0,Y 153.167,Z 471.306,A -85,B 0,C 180,E1 -26849.332,E2 -26849.332} C_VEL
LIN {X 0,Y 147.586,Z 483.494,A -85,B 0,C 180,E1 -26851.003,E2 -26851.003} C_VEL
LIN {X 0,Y 141.29,Z 495.1,A -85,B 0,C 180,E1 -26853.173,E2 -26853.173} C_VEL
LIN {X 0,Y 134.398,Z 505.893,A -85,B 0,C 180,E1 -26855.853,E2 -26855.853} C_VEL
LIN {X 0,Y 126.814,Z 515.936,A -85,B 0,C 180,E1 -26859.117,E2 -26859.117} C_VEL
LIN {X 0,Y 119.831,Z 524.272,A -85,B 0,C 180,E1 -26862.853,E2 -26862.853} C_VEL
LIN {X 0,Y 112.272,Z 532.236,A -85,B 0,C 180,E1 -26867.707,E2 -26867.707} C_VEL
LIN {X 0,Y 105.726,Z 538.643,A -85,B 0,C 180,E1 -26873.255,E2 -26873.255} C_VEL
LIN {X 0,Y 99.588,Z 544.321,A -85,B 0,C 180,E1 -26880.397,E2 -26880.397} C_VEL
LIN {X 0,Y 94.901,Z 548.445,A -85,B 0,C 180,E1 -26888.267,E2 -26888.267} C_VEL
LIN {X 0,Y 92.104,Z 551.136,A -85,B 0,C 180,E1 -26896.767,E2 -26896.767} C_VEL
LIN {X 0,Y 90.892,Z 552.477,A -85,B 0,C 180,E1 -26905.565,E2 -26905.565} C_VEL
LIN {X 0,Y 90.914,Z 552.651,A -85,B 0,C 180,E1 -26910,E2 -26910} C_VEL
LIN {X 0,Y 91.312,Z 552.016,A -85,B 0,C 180,E1 -26918.855,E2 -26918.855} C_VEL
LIN {X 0,Y 93.277,Z 550.044,A -85,B 0,C 180,E1 -26927.54,E2 -26927.54} C_VEL
LIN {X 0,Y 96.952,Z 546.691,A -85,B 0,C 180,E1 -26935.78,E2 -26935.78} C_VEL
LIN {X 0,Y 102.43,Z 541.854,A -85,B 0,C 180,E1 -26943.291,E2 -26943.291} C_VEL
LIN {X 0,Y 107.606,Z 537.018,A -85,B 0,C 180,E1 -26948.568,E2 -26948.568} C_VEL
LIN {X 0,Y 114.284,Z 530.394,A -85,B 0,C 180,E1 -26953.773,E2 -26953.773} C_VEL
LIN {X 0,Y 122.043,Z 521.959,A -85,B 0,C 180,E1 -26958.469,E2 -26958.469} C_VEL
LIN {X 0,Y 129.233,Z 513.154,A -85,B 0,C 180,E1 -26962.048,E2 -26962.048} C_VEL
LIN {X 0,Y 136.88,Z 502.484,A -85,B 0,C 180,E1 -26965.234,E2 -26965.234} C_VEL
LIN {X 0,Y 143.459,Z 491.688,A -85,B 0,C 180,E1 -26967.677,E2 -26967.677} C_VEL
LIN {X 0,Y 149.596,Z 479.871,A -85,B 0,C 180,E1 -26969.681,E2 -26969.681} C_VEL
LIN {X 0,Y 155.225,Z 466.82,A -85,B 0,C 180,E1 -26971.307,E2 -26971.307} C_VEL
LIN {X 0,Y 159.775,Z 453.387,A -85,B 0,C 180,E1 -26972.533,E2 -26972.533} C_VEL
LIN {X 0,Y 163.437,Z 438.744,A -85,B 0,C 180,E1 -26973.446,E2 -26973.446} C_VEL
LIN {X 0,Y 165.719,Z 424.485,A -85,B 0,C 180,E1 -26974.063,E2 -26974.063} C_VEL
LIN {X 0,Y 168.657,Z 395.129,A -85,B 0,C 180,E1 -26974.887,E2 -26974.887} C_VEL
LIN {X 0,Y 165.316,Z 387.521,A -85,B 0,C 180,E1 -26978.352,E2 -26978.352} C_VEL
LIN {X 0,Y 162.448,Z 381.803,A -85,B 0,C 180,E1 -26981.85,E2 -26981.85} C_VEL
LIN {X 0,Y 160.797,Z 378.768,A -85,B 0,C 180,E1 -26984.229,E2 -26984.229} C_VEL
LIN {X 0,Y 159.245,Z 375.763,A -85,B 0,C 180,E1 -26986.927,E2 -26986.927} C_VEL
LIN {X 0,Y 157.603,Z 372.471,A -85,B 0,C 180,E1 -26990.697,E2 -26990.697} C_VEL
LIN {X 0,Y 156.064,Z 368.286,A -85,B 0,C 180,E1 -27000,E2 -27000} C_VEL
LIN {X 0,Y 157.755,Z 372.727,A -85,B 0,C 180,E1 -27009.617,E2 -27009.617} C_VEL
LIN {X 0,Y 159.793,Z 376.8,A -85,B 0,C 180,E1 -27013.999,E2 -27013.999} C_VEL
LIN {X 0,Y 162.098,Z 381.151,A -85,B 0,C 180,E1 -27017.588,E2 -27017.588} C_VEL
LIN {X 0,Y 164.498,Z 385.866,A -85,B 0,C 180,E1 -27020.63,E2 -27020.63} C_VEL
LIN {X 0,Y 167.142,Z 391.792,A -85,B 0,C 180,E1 -27023.544,E2 -27023.544} C_VEL
LIN {X 0,Y 168.577,Z 396.09,A -85,B 0,C 180,E1 -27025.063,E2 -27025.063} C_VEL
LIN {X 0,Y 165.146,Z 429.786,A -85,B 0,C 180,E1 -27026.068,E2 -27026.068} C_VEL
LIN {X 0,Y 162.36,Z 444.36,A -85,B 0,C 180,E1 -27026.729,E2 -27026.729} C_VEL
LIN {X 0,Y 158.273,Z 458.901,A -85,B 0,C 180,E1 -27027.713,E2 -27027.713} C_VEL
LIN {X 0,Y 153.603,Z 471.628,A -85,B 0,C 180,E1 -27028.952,E2 -27028.952} C_VEL
LIN {X 0,Y 147.965,Z 484.04,A -85,B 0,C 180,E1 -27030.585,E2 -27030.585} C_VEL
LIN {X 0,Y 141.775,Z 495.39,A -85,B 0,C 180,E1 -27032.575,E2 -27032.575} C_VEL
LIN {X 0,Y 134.599,Z 506.744,A -85,B 0,C 180,E1 -27035.293,E2 -27035.293} C_VEL
LIN {X 0,Y 127.627,Z 516.21,A -85,B 0,C 180,E1 -27038.309,E2 -27038.309} C_VEL
LIN {X 0,Y 120.423,Z 524.776,A -85,B 0,C 180,E1 -27041.92,E2 -27041.92} C_VEL
LIN {X 0,Y 112.803,Z 532.974,A -85,B 0,C 180,E1 -27046.74,E2 -27046.74} C_VEL
LIN {X 0,Y 106.978,Z 538.723,A -85,B 0,C 180,E1 -27051.385,E2 -27051.385} C_VEL
LIN {X 0,Y 102.027,Z 543.428,A -85,B 0,C 180,E1 -27056.561,E2 -27056.561} C_VEL
LIN {X 0,Y 96.619,Z 548.304,A -85,B 0,C 180,E1 -27064.124,E2 -27064.124} C_VEL
LIN {X 0,Y 92.945,Z 551.695,A -85,B 0,C 180,E1 -27072.395,E2 -27072.395} C_VEL
LIN {X 0,Y 91.137,Z 553.699,A -85,B 0,C 180,E1 -27081.128,E2 -27081.128} C_VEL
LIN {X 0,Y 90.84,Z 554.356,A -85,B 0,C 180,E1 -27090,E2 -27090} C_VEL
LIN {X 0,Y 91.139,Z 553.671,A -85,B 0,C 180,E1 -27098.872,E2 -27098.872} C_VEL
LIN {X 0,Y 92.96,Z 551.643,A -85,B 0,C 180,E1 -27107.602,E2 -27107.602} C_VEL
LIN {X 0,Y 96.617,Z 548.225,A -85,B 0,C 180,E1 -27115.877,E2 -27115.877} C_VEL
LIN {X 0,Y 101.957,Z 543.314,A -85,B 0,C 180,E1 -27123.466,E2 -27123.466} C_VEL
LIN {X 0,Y 106.96,Z 538.579,A -85,B 0,C 180,E1 -27128.624,E2 -27128.624} C_VEL
LIN {X 0,Y 113.818,Z 531.719,A -85,B 0,C 180,E1 -27133.999,E2 -27133.999} C_VEL
LIN {X 0,Y 121.541,Z 523.205,A -85,B 0,C 180,E1 -27138.738,E2 -27138.738} C_VEL
LIN {X 0,Y 128.87,Z 514.322,A -85,B 0,C 180,E1 -27142.256,E2 -27142.256} C_VEL
LIN {X 0,Y 136.507,Z 503.56,A -85,B 0,C 180,E1 -27145.46,E2 -27145.46} C_VEL
LIN {X 0,Y 139.848,Z 498.27,A -85,B 0,C 180,E1 -27146.724,E2 -27146.724} C_VEL
LIN {X 0,Y 142.19,Z 493.721,A -85,B 0,C 180,E1 -27147.933,E2 -27147.933} C_VEL
LIN {X 0,Y 144.893,Z 486.142,A -85,B 0,C 180,E1 -27150.252,E2 -27150.252} C_VEL
LIN {X 0,Y 147.436,Z 478.203,A -85,B 0,C 180,E1 -27152.339,E2 -27152.339} C_VEL
LIN {X 0,Y 149.43,Z 473.097,A -85,B 0,C 180,E1 -27153.176,E2 -27153.176} C_VEL
LIN {X 0,Y 154.384,Z 460.345,A -85,B 0,C 180,E1 -27154.41,E2 -27154.41} C_VEL
LIN {X 0,Y 158.559,Z 446.121,A -85,B 0,C 180,E1 -27155.422,E2 -27155.422} C_VEL
LIN {X 0,Y 161.671,Z 431.162,A -85,B 0,C 180,E1 -27156.076,E2 -27156.076} C_VEL
LIN {X 0,Y 164.201,Z 408.388,A -85,B 0,C 180,E1 -27156.778,E2 -27156.778} C_VEL
LIN {X 0,Y 165.111,Z 398.943,A -85,B 0,C 180,E1 -27157.064,E2 -27157.064} C_VEL
LIN {X 0,Y 163.812,Z 395.201,A -85,B 0,C 180,E1 -27158.592,E2 -27158.592} C_VEL
LIN {X 0,Y 161.056,Z 388.95,A -85,B 0,C 180,E1 -27162.102,E2 -27162.102} C_VEL
LIN {X 0,Y 159.089,Z 385.114,A -85,B 0,C 180,E1 -27165.072,E2 -27165.072} C_VEL
LIN {X 0,Y 157.645,Z 382.166,A -85,B 0,C 180,E1 -27167.775,E2 -27167.775} C_VEL
LIN {X 0,Y 156.239,Z 379.127,A -85,B 0,C 180,E1 -27171.268,E2 -27171.268} C_VEL
LIN {X 0,Y 154.89,Z 375.171,A -85,B 0,C 180,E1 -27179.35,E2 -27179.35} C_VEL
LIN {X 0,Y 154.888,Z 375.364,A -85,B 0,C 180,E1 -27181.3,E2 -27181.3} C_VEL
LIN {X 0,Y 156.525,Z 379.771,A -85,B 0,C 180,E1 -27189.734,E2 -27189.734} C_VEL
LIN {X 0,Y 158.356,Z 383.598,A -85,B 0,C 180,E1 -27193.801,E2 -27193.801} C_VEL
LIN {X 0,Y 160.223,Z 387.359,A -85,B 0,C 180,E1 -27196.894,E2 -27196.894} C_VEL
LIN {X 0,Y 162.526,Z 392.199,A -85,B 0,C 180,E1 -27200.025,E2 -27200.025} C_VEL
LIN {X 0,Y 165.18,Z 398.432,A -85,B 0,C 180,E1 -27203.114,E2 -27203.114} C_VEL
LIN {X 0,Y 161.927,Z 428.835,A -85,B 0,C 180,E1 -27203.988,E2 -27203.988} C_VEL
LIN {X 0,Y 159.11,Z 443.196,A -85,B 0,C 180,E1 -27204.637,E2 -27204.637} C_VEL
LIN {X 0,Y 154.93,Z 457.827,A -85,B 0,C 180,E1 -27205.636,E2 -27205.636} C_VEL
LIN {X 0,Y 149.818,Z 471.378,A -85,B 0,C 180,E1 -27206.966,E2 -27206.966} C_VEL
LIN {X 0,Y 144.063,Z 483.565,A -85,B 0,C 180,E1 -27208.586,E2 -27208.586} C_VEL
LIN {X 0,Y 137.657,Z 494.934,A -85,B 0,C 180,E1 -27210.633,E2 -27210.633} C_VEL
LIN {X 0,Y 130.366,Z 505.963,A -85,B 0,C 180,E1 -27213.323,E2 -27213.323} C_VEL
LIN {X 0,Y 122.45,Z 516.005,A -85,B 0,C 180,E1 -27216.533,E2 -27216.533} C_VEL
LIN {X 0,Y 115.093,Z 524.341,A -85,B 0,C 180,E1 -27220.246,E2 -27220.246} C_VEL
LIN {X 0,Y 107.103,Z 532.305,A -85,B 0,C 180,E1 -27225.139,E2 -27225.139} C_VEL
LIN {X 0,Y 100.085,Z 538.711,A -85,B 0,C 180,E1 -27230.804,E2 -27230.804} C_VEL
LIN {X 0,Y 93.466,Z 544.389,A -85,B 0,C 180,E1 -27238.241,E2 -27238.241} C_VEL
LIN {X 0,Y 88.306,Z 548.513,A -85,B 0,C 180,E1 -27246.551,E2 -27246.551} C_VEL
LIN {X 0,Y 85.201,Z 551.203,A -85,B 0,C 180,E1 -27255.673,E2 -27255.673} C_VEL
LIN {X 0,Y 83.812,Z 552.544,A -85,B 0,C 180,E1 -27265.19,E2 -27265.19} C_VEL
LIN {X 0,Y 83.813,Z 552.718,A -85,B 0,C 180,E1 -27270,E2 -27270} C_VEL
LIN {X 0,Y 84.295,Z 552.082,A -85,B 0,C 180,E1 -27279.598,E2 -27279.598} C_VEL
LIN {X 0,Y 86.494,Z 550.111,A -85,B 0,C 180,E1 -27288.966,E2 -27288.966} C_VEL
LIN {X 0,Y 90.597,Z 546.757,A -85,B 0,C 180,E1 -27297.738,E2 -27297.738} C_VEL
LIN {X 0,Y 96.546,Z 541.919,A -85,B 0,C 180,E1 -27305.615,E2 -27305.615} C_VEL
LIN {X 0,Y 101.759,Z 537.429,A -85,B 0,C 180,E1 -27310.741,E2 -27310.741} C_VEL
LIN {X 0,Y 109.255,Z 530.459,A -85,B 0,C 180,E1 -27316.357,E2 -27316.357} C_VEL
LIN {X 0,Y 117.438,Z 522.023,A -85,B 0,C 180,E1 -27321.073,E2 -27321.073} C_VEL
LIN {X 0,Y 124.994,Z 513.218,A -85,B 0,C 180,E1 -27324.613,E2 -27324.613} C_VEL
LIN {X 0,Y 132.944,Z 502.547,A -85,B 0,C 180,E1 -27327.758,E2 -27327.758} C_VEL
LIN {X 0,Y 139.783,Z 491.751,A -85,B 0,C 180,E1 -27330.143,E2 -27330.143} C_VEL
LIN {X 0,Y 146.146,Z 479.933,A -85,B 0,C 180,E1 -27332.081,E2 -27332.081} C_VEL
LIN {X 0,Y 151.94,Z 466.881,A -85,B 0,C 180,E1 -27333.659,E2 -27333.659} C_VEL
LIN {X 0,Y 156.566,Z 453.676,A -85,B 0,C 180,E1 -27334.816,E2 -27334.816} C_VEL
LIN {X 0,Y 160.321,Z 439.149,A -85,B 0,C 180,E1 -27335.696,E2 -27335.696} C_VEL
LIN {X 0,Y 162.637,Z 425.376,A -85,B 0,C 180,E1 -27336.285,E2 -27336.285} C_VEL
LIN {X 0,Y 165.438,Z 398.675,A -85,B 0,C 180,E1 -27336.997,E2 -27336.997} C_VEL
LIN {X 0,Y 162.296,Z 391.332,A -85,B 0,C 180,E1 -27340.719,E2 -27340.719} C_VEL
LIN {X 0,Y 159.76,Z 386.038,A -85,B 0,C 180,E1 -27344.369,E2 -27344.369} C_VEL
LIN {X 0,Y 157.845,Z 382.269,A -85,B 0,C 180,E1 -27347.872,E2 -27347.872} C_VEL
LIN {X 0,Y 156.363,Z 379.191,A -85,B 0,C 180,E1 -27351.656,E2 -27351.656} C_VEL
LIN {X 0,Y 155.189,Z 375.413,A -85,B 0,C 180,E1 -27360,E2 -27360} C_VEL
LIN {X 0,Y 156.68,Z 379.703,A -85,B 0,C 180,E1 -27369.162,E2 -27369.162} C_VEL
LIN {X 0,Y 158.529,Z 383.676,A -85,B 0,C 180,E1 -27373.418,E2 -27373.418} C_VEL
LIN {X 0,Y 160.45,Z 387.476,A -85,B 0,C 180,E1 -27376.625,E2 -27376.625} C_VEL
LIN {X 0,Y 162.703,Z 392.286,A -85,B 0,C 180,E1 -27379.722,E2 -27379.722} C_VEL
LIN {X 0,Y 164.785,Z 397.347,A -85,B 0,C 180,E1 -27382.225,E2 -27382.225} C_VEL
LIN {X 0,Y 165.409,Z 399.26,A -85,B 0,C 180,E1 -27382.956,E2 -27382.956} C_VEL
LIN {X 0,Y 162.063,Z 430.286,A -85,B 0,C 180,E1 -27383.835,E2 -27383.835} C_VEL
LIN {X 0,Y 159.223,Z 444.596,A -85,B 0,C 180,E1 -27384.466,E2 -27384.466} C_VEL
LIN {X 0,Y 155.088,Z 458.841,A -85,B 0,C 180,E1 -27385.382,E2 -27385.382} C_VEL
LIN {X 0,Y 150.291,Z 471.567,A -85,B 0,C 180,E1 -27386.58,E2 -27386.58} C_VEL
LIN {X 0,Y 144.483,Z 483.978,A -85,B 0,C 180,E1 -27388.162,E2 -27388.162} C_VEL
LIN {X 0,Y 138.08,Z 495.327,A -85,B 0,C 180,E1 -27390.089,E2 -27390.089} C_VEL
LIN {X 0,Y 131.093,Z 505.993,A -85,B 0,C 180,E1 -27392.567,E2 -27392.567} C_VEL
LIN {X 0,Y 123.342,Z 516.145,A -85,B 0,C 180,E1 -27395.714,E2 -27395.714} C_VEL
LIN {X 0,Y 115.778,Z 524.711,A -85,B 0,C 180,E1 -27399.292,E2 -27399.292} C_VEL
LIN {X 0,Y 107.7,Z 532.908,A -85,B 0,C 180,E1 -27404.128,E2 -27404.128} C_VEL
LIN {X 0,Y 101.485,Z 538.657,A -85,B 0,C 180,E1 -27408.862,E2 -27408.862} C_VEL
LIN {X 0,Y 94.512,Z 544.75,A -85,B 0,C 180,E1 -27416.104,E2 -27416.104} C_VEL
LIN {X 0,Y 90.249,Z 548.238,A -85,B 0,C 180,E1 -27422.146,E2 -27422.146} C_VEL
LIN {X 0,Y 86.178,Z 551.628,A -85,B 0,C 180,E1 -27430.962,E2 -27430.962} C_VEL
LIN {X 0,Y 84.123,Z 553.632,A -85,B 0,C 180,E1 -27440.382,E2 -27440.382} C_VEL
LIN {X 0,Y 83.761,Z 554.29,A -85,B 0,C 180,E1 -27450,E2 -27450} C_VEL
LIN {X 0,Y 84.125,Z 553.604,A -85,B 0,C 180,E1 -27459.618,E2 -27459.618} C_VEL
LIN {X 0,Y 86.191,Z 551.575,A -85,B 0,C 180,E1 -27469.036,E2 -27469.036} C_VEL
LIN {X 0,Y 90.245,Z 548.157,A -85,B 0,C 180,E1 -27477.856,E2 -27477.856} C_VEL
LIN {X 0,Y 96.057,Z 543.245,A -85,B 0,C 180,E1 -27485.825,E2 -27485.825} C_VEL
LIN {X 0,Y 103.465,Z 536.698,A -85,B 0,C 180,E1 -27492.785,E2 -27492.785} C_VEL
LIN {X 0,Y 111.073,Z 529.415,A -85,B 0,C 180,E1 -27498.026,E2 -27498.026} C_VEL
LIN {X 0,Y 118.215,Z 521.78,A -85,B 0,C 180,E1 -27501.972,E2 -27501.972} C_VEL
LIN {X 0,Y 125.94,Z 512.624,A -85,B 0,C 180,E1 -27505.396,E2 -27505.396} C_VEL
LIN {X 0,Y 132.602,Z 503.491,A -85,B 0,C 180,E1 -27507.994,E2 -27507.994} C_VEL
LIN {X 0,Y 139.469,Z 492.593,A -85,B 0,C 180,E1 -27510.369,E2 -27510.369} C_VEL
LIN {X 0,Y 145.938,Z 480.66,A -85,B 0,C 180,E1 -27512.236,E2 -27512.236} C_VEL
LIN {X 0,Y 149.43,Z 473.097,A -85,B 0,C 180,E1 -27513.176,E2 -27513.176} C_VEL
LIN {X 0,Y 151.301,Z 467.878,A -85,B 0,C 180,E1 -27513.964,E2 -27513.964} C_VEL
LIN {X 0,Y 153.21,Z 459.317,A -85,B 0,C 180,E1 -27515.72,E2 -27515.72} C_VEL
LIN {X 0,Y 154.803,Z 450.522,A -85,B 0,C 180,E1 -27517.309,E2 -27517.309} C_VEL
LIN {X 0,Y 156.023,Z 444.942,A -85,B 0,C 180,E1 -27517.852,E2 -27517.852} C_VEL
LIN {X 0,Y 158.936,Z 431.021,A -85,B 0,C 180,E1 -27518.418,E2 -27518.418} C_VEL
LIN {X 0,Y 161.656,Z 407.202,A -85,B 0,C 180,E1 -27519.113,E2 -27519.113} C_VEL
LIN {X 0,Y 162.128,Z 402.16,A -85,B 0,C 180,E1 -27519.29,E2 -27519.29} C_VEL
LIN {X 0,Y 159.775,Z 396.242,A -85,B 0,C 180,E1 -27522.48,E2 -27522.48} C_VEL
LIN {X 0,Y 157.678,Z 391.715,A -85,B 0,C 180,E1 -27525.867,E2 -27525.867} C_VEL
LIN {X 0,Y 156.305,Z 388.733,A -85,B 0,C 180,E1 -27528.669,E2 -27528.669} C_VEL
LIN {X 0,Y 155.144,Z 385.994,A -85,B 0,C 180,E1 -27531.862,E2 -27531.862} C_VEL
LIN {X 0,Y 154.025,Z 382.112,A -85,B 0,C 180,E1 -27540,E2 -27540} C_VEL
LIN {X 0,Y 154.153,Z 383.872,A -85,B 0,C 180,E1 -27543.922,E2 -27543.922} C_VEL
LIN {X 0,Y 155.393,Z 386.612,A -85,B 0,C 180,E1 -27549.108,E2 -27549.108} C_VEL
LIN {X 0,Y 157.008,Z 390.26,A -85,B 0,C 180,E1 -27553.023,E2 -27553.023} C_VEL
LIN {X 0,Y 158.803,Z 394.138,A -85,B 0,C 180,E1 -27556.223,E2 -27556.223} C_VEL
LIN {X 0,Y 161.189,Z 399.596,A -85,B 0,C 180,E1 -27559.659,E2 -27559.659} C_VEL
LIN {X 0,Y 162.167,Z 402.047,A -85,B 0,C 180,E1 -27560.909,E2 -27560.909} C_VEL
LIN {X 0,Y 159.169,Z 428.993,A -85,B 0,C 180,E1 -27561.664,E2 -27561.664} C_VEL
LIN {X 0,Y 156.286,Z 443.267,A -85,B 0,C 180,E1 -27562.27,E2 -27562.27} C_VEL
LIN {X 0,Y 152.368,Z 456.772,A -85,B 0,C 180,E1 -27563.132,E2 -27563.132} C_VEL
LIN {X 0,Y 147.489,Z 469.685,A -85,B 0,C 180,E1 -27564.313,E2 -27564.313} C_VEL
LIN {X 0,Y 141.533,Z 482.212,A -85,B 0,C 180,E1 -27565.842,E2 -27565.842} C_VEL
LIN {X 0,Y 135.01,Z 493.634,A -85,B 0,C 180,E1 -27567.758,E2 -27567.758} C_VEL
LIN {X 0,Y 127.996,Z 504.121,A -85,B 0,C 180,E1 -27570.142,E2 -27570.142} C_VEL
LIN {X 0,Y 119.713,Z 514.542,A -85,B 0,C 180,E1 -27573.222,E2 -27573.222} C_VEL
LIN {X 0,Y 111.892,Z 523.134,A -85,B 0,C 180,E1 -27576.791,E2 -27576.791} C_VEL
LIN {X 0,Y 103.324,Z 531.367,A -85,B 0,C 180,E1 -27581.566,E2 -27581.566} C_VEL
LIN {X 0,Y 95.029,Z 538.455,A -85,B 0,C 180,E1 -27587.695,E2 -27587.695} C_VEL
LIN {X 0,Y 89.162,Z 543.219,A -85,B 0,C 180,E1 -27593.76,E2 -27593.76} C_VEL
LIN {X 0,Y 84.391,Z 546.705,A -85,B 0,C 180,E1 -27600.022,E2 -27600.022} C_VEL
LIN {X 0,Y 79.792,Z 550.098,A -85,B 0,C 180,E1 -27609.371,E2 -27609.371} C_VEL
LIN {X 0,Y 77.296,Z 552.106,A -85,B 0,C 180,E1 -27619.523,E2 -27619.523} C_VEL
LIN {X 0,Y 76.735,Z 552.784,A -85,B 0,C 180,E1 -27630,E2 -27630} C_VEL
LIN {X 0,Y 77.29,Z 552.148,A -85,B 0,C 180,E1 -27640.478,E2 -27640.478} C_VEL
LIN {X 0,Y 79.776,Z 550.177,A -85,B 0,C 180,E1 -27650.632,E2 -27650.632} C_VEL
LIN {X 0,Y 84.369,Z 546.823,A -85,B 0,C 180,E1 -27659.986,E2 -27659.986} C_VEL
LIN {X 0,Y 90.845,Z 541.985,A -85,B 0,C 180,E1 -27668.234,E2 -27668.234} C_VEL
LIN {X 0,Y 98.768,Z 535.51,A -85,B 0,C 180,E1 -27675.361,E2 -27675.361} C_VEL
LIN {X 0,Y 106.839,Z 528.297,A -85,B 0,C 180,E1 -27680.616,E2 -27680.616} C_VEL
LIN {X 0,Y 114.367,Z 520.737,A -85,B 0,C 180,E1 -27684.509,E2 -27684.509} C_VEL
LIN {X 0,Y 122.365,Z 511.658,A -85,B 0,C 180,E1 -27687.902,E2 -27687.902} C_VEL
LIN {X 0,Y 130.386,Z 501.045,A -85,B 0,C 180,E1 -27690.837,E2 -27690.837} C_VEL
LIN {X 0,Y 137.818,Z 489.428,A -85,B 0,C 180,E1 -27693.175,E2 -27693.175} C_VEL
LIN {X 0,Y 144.451,Z 477.002,A -85,B 0,C 180,E1 -27694.978,E2 -27694.978} C_VEL
LIN {X 0,Y 149.679,Z 465.023,A -85,B 0,C 180,E1 -27696.287,E2 -27696.287} C_VEL
LIN {X 0,Y 154.219,Z 451.945,A -85,B 0,C 180,E1 -27697.319,E2 -27697.319} C_VEL
LIN {X 0,Y 157.872,Z 437.584,A -85,B 0,C 180,E1 -27698.121,E2 -27698.121} C_VEL
LIN {X 0,Y 160.144,Z 423.754,A -85,B 0,C 180,E1 -27698.643,E2 -27698.643} C_VEL
LIN {X 0,Y 162.42,Z 402.343,A -85,B 0,C 180,E1 -27699.204,E2 -27699.204} C_VEL
LIN {X 0,Y 159.974,Z 396.358,A -85,B 0,C 180,E1 -27702.513,E2 -27702.513} C_VEL
LIN {X 0,Y 157.923,Z 391.92,A -85,B 0,C 180,E1 -27705.851,E2 -27705.851} C_VEL
LIN {X 0,Y 156.49,Z 388.757,A -85,B 0,C 180,E1 -27708.832,E2 -27708.832} C_VEL
LIN {X 0,Y 155.302,Z 386.074,A -85,B 0,C 180,E1 -27712.197,E2 -27712.197} C_VEL
LIN {X 0,Y 154.314,Z 382.534,A -85,B 0,C 180,E1 -27720,E2 -27720} C_VEL
LIN {X 0,Y 155.6,Z 386.608,A -85,B 0,C 180,E1 -27728.645,E2 -27728.645} C_VEL
LIN {X 0,Y 157.247,Z 390.438,A -85,B 0,C 180,E1 -27732.749,E2 -27732.749} C_VEL
LIN {X 0,Y 159.12,Z 394.428,A -85,B 0,C 180,E1 -27736.089,E2 -27736.089} C_VEL
LIN {X 0,Y 161.453,Z 399.899,A -85,B 0,C 180,E1 -27739.467,E2 -27739.467} C_VEL
LIN {X 0,Y 162.417,Z 402.492,A -85,B 0,C 180,E1 -27740.724,E2 -27740.724} C_VEL
LIN {X 0,Y 159.301,Z 430.428,A -85,B 0,C 180,E1 -27741.513,E2 -27741.513} C_VEL
LIN {X 0,Y 156.293,Z 445.043,A -85,B 0,C 180,E1 -27742.128,E2 -27742.128} C_VEL
LIN {X 0,Y 152.183,Z 458.782,A -85,B 0,C 180,E1 -27742.969,E2 -27742.969} C_VEL
LIN {X 0,Y 147.25,Z 471.506,A -85,B 0,C 180,E1 -27744.108,E2 -27744.108} C_VEL
LIN {X 0,Y 141.267,Z 483.916,A -85,B 0,C 180,E1 -27745.619,E2 -27745.619} C_VEL
LIN {X 0,Y 134.646,Z 495.264,A -85,B 0,C 180,E1 -27747.463,E2 -27747.463} C_VEL
LIN {X 0,Y 126.921,Z 506.603,A -85,B 0,C 180,E1 -27750.04,E2 -27750.04} C_VEL
LIN {X 0,Y 119.331,Z 516.081,A -85,B 0,C 180,E1 -27752.941,E2 -27752.941} C_VEL
LIN {X 0,Y 111.401,Z 524.647,A -85,B 0,C 180,E1 -27756.453,E2 -27756.453} C_VEL
LIN {X 0,Y 102.864,Z 532.843,A -85,B 0,C 180,E1 -27761.276,E2 -27761.276} C_VEL
LIN {X 0,Y 96.219,Z 538.592,A -85,B 0,C 180,E1 -27766.062,E2 -27766.062} C_VEL
LIN {X 0,Y 90.418,Z 543.296,A -85,B 0,C 180,E1 -27771.552,E2 -27771.552} C_VEL
LIN {X 0,Y 84.007,Z 548.172,A -85,B 0,C 180,E1 -27779.872,E2 -27779.872} C_VEL
LIN {X 0,Y 79.462,Z 551.562,A -85,B 0,C 180,E1 -27789.282,E2 -27789.282} C_VEL
LIN {X 0,Y 77.111,Z 553.566,A -85,B 0,C 180,E1 -27799.498,E2 -27799.498} C_VEL
LIN {X 0,Y 76.673,Z 554.223,A -85,B 0,C 180,E1 -27810,E2 -27810} C_VEL
LIN {X 0,Y 77.113,Z 553.537,A -85,B 0,C 180,E1 -27820.503,E2 -27820.503} C_VEL
LIN {X 0,Y 79.473,Z 551.508,A -85,B 0,C 180,E1 -27830.716,E2 -27830.716} C_VEL
LIN {X 0,Y 84.002,Z 548.089,A -85,B 0,C 180,E1 -27840.131,E2 -27840.131} C_VEL
LIN {X 0,Y 90.348,Z 543.177,A -85,B 0,C 180,E1 -27848.484,E2 -27848.484} C_VEL
LIN {X 0,Y 96.21,Z 538.442,A -85,B 0,C 180,E1 -27853.943,E2 -27853.943} C_VEL
LIN {X 0,Y 104.038,Z 531.582,A -85,B 0,C 180,E1 -27859.46,E2 -27859.46} C_VEL
LIN {X 0,Y 112.658,Z 523.067,A -85,B 0,C 180,E1 -27864.191,E2 -27864.191} C_VEL
LIN {X 0,Y 120.686,Z 514.184,A -85,B 0,C 180,E1 -27867.605,E2 -27867.605} C_VEL
LIN {X 0,Y 128.969,Z 503.421,A -85,B 0,C 180,E1 -27870.678,E2 -27870.678} C_VEL
LIN {X 0,Y 136.084,Z 492.522,A -85,B 0,C 180,E1 -27872.981,E2 -27872.981} C_VEL
LIN {X 0,Y 142.771,Z 480.589,A -85,B 0,C 180,E1 -27874.757,E2 -27874.757} C_VEL
LIN {X 0,Y 148.785,Z 467.352,A -85,B 0,C 180,E1 -27876.232,E2 -27876.232} C_VEL
LIN {X 0,Y 153.759,Z 453.199,A -85,B 0,C 180,E1 -27877.349,E2 -27877.349} C_VEL
LIN {X 0,Y 156.023,Z 444.942,A -85,B 0,C 180,E1 -27877.852,E2 -27877.852} C_VEL
LIN {X 0,Y 157.129,Z 439.285,A -85,B 0,C 180,E1 -27878.335,E2 -27878.335} C_VEL
LIN {X 0,Y 157.816,Z 430.07,A -85,B 0,C 180,E1 -27879.652,E2 -27879.652} C_VEL
LIN {X 0,Y 158.049,Z 420.761,A -85,B 0,C 180,E1 -27880.914,E2 -27880.914} C_VEL
LIN {X 0,Y 158.433,Z 414.951,A -85,B 0,C 180,E1 -27881.302,E2 -27881.302} C_VEL
LIN {X 0,Y 159.344,Z 405.852,A -85,B 0,C 180,E1 -27881.588,E2 -27881.588} C_VEL
LIN {X 0,Y 157.341,Z 400.73,A -85,B 0,C 180,E1 -27884.753,E2 -27884.753} C_VEL
LIN {X 0,Y 155.354,Z 395.947,A -85,B 0,C 180,E1 -27888.757,E2 -27888.757} C_VEL
LIN {X 0,Y 154.068,Z 392.851,A -85,B 0,C 180,E1 -27892.464,E2 -27892.464} C_VEL
LIN {X 0,Y 153.16,Z 389.155,A -85,B 0,C 180,E1 -27900,E2 -27900} C_VEL
LIN {X 0,Y 154.296,Z 393.462,A -85,B 0,C 180,E1 -27908.513,E2 -27908.513} C_VEL
LIN {X 0,Y 155.75,Z 397.051,A -85,B 0,C 180,E1 -27912.362,E2 -27912.362} C_VEL
LIN {X 0,Y 157.349,Z 400.763,A -85,B 0,C 180,E1 -27915.441,E2 -27915.441} C_VEL
LIN {X 0,Y 159.367,Z 405.861,A -85,B 0,C 180,E1 -27918.614,E2 -27918.614} C_VEL
LIN {X 0,Y 156.526,Z 429.958,A -85,B 0,C 180,E1 -27919.271,E2 -27919.271} C_VEL
LIN {X 0,Y 153.445,Z 444.493,A -85,B 0,C 180,E1 -27919.884,E2 -27919.884} C_VEL
LIN {X 0,Y 149.339,Z 457.974,A -85,B 0,C 180,E1 -27920.721,E2 -27920.721} C_VEL
LIN {X 0,Y 143.942,Z 471.522,A -85,B 0,C 180,E1 -27921.927,E2 -27921.927} C_VEL
LIN {X 0,Y 137.84,Z 483.707,A -85,B 0,C 180,E1 -27923.402,E2 -27923.402} C_VEL
LIN {X 0,Y 130.675,Z 495.54,A -85,B 0,C 180,E1 -27925.359,E2 -27925.359} C_VEL
LIN {X 0,Y 123.139,Z 506.102,A -85,B 0,C 180,E1 -27927.794,E2 -27927.794} C_VEL
LIN {X 0,Y 114.563,Z 516.143,A -85,B 0,C 180,E1 -27930.814,E2 -27930.814} C_VEL
LIN {X 0,Y 106.447,Z 524.479,A -85,B 0,C 180,E1 -27934.383,E2 -27934.383} C_VEL
LIN {X 0,Y 97.517,Z 532.442,A -85,B 0,C 180,E1 -27939.219,E2 -27939.219} C_VEL
LIN {X 0,Y 89.452,Z 538.848,A -85,B 0,C 180,E1 -27945.001,E2 -27945.001} C_VEL
LIN {X 0,Y 81.707,Z 544.525,A -85,B 0,C 180,E1 -27952.98,E2 -27952.98} C_VEL
LIN {X 0,Y 75.422,Z 548.648,A -85,B 0,C 180,E1 -27962.231,E2 -27962.231} C_VEL
LIN {X 0,Y 71.476,Z 551.338,A -85,B 0,C 180,E1 -27972.844,E2 -27972.844} C_VEL
LIN {X 0,Y 69.674,Z 552.677,A -85,B 0,C 180,E1 -27984.211,E2 -27984.211} C_VEL
LIN {X 0,Y 69.647,Z 552.851,A -85,B 0,C 180,E1 -27990,E2 -27990} C_VEL
LIN {X 0,Y 70.317,Z 552.215,A -85,B 0,C 180,E1 -28001.53,E2 -28001.53} C_VEL
LIN {X 0,Y 73.146,Z 550.243,A -85,B 0,C 180,E1 -28012.601,E2 -28012.601} C_VEL
LIN {X 0,Y 78.29,Z 546.889,A -85,B 0,C 180,E1 -28022.588,E2 -28022.588} C_VEL
LIN {X 0,Y 85.362,Z 542.051,A -85,B 0,C 180,E1 -28031.196,E2 -28031.196} C_VEL
LIN {X 0,Y 93.893,Z 535.576,A -85,B 0,C 180,E1 -28038.46,E2 -28038.46} C_VEL
LIN {X 0,Y 102.471,Z 528.362,A -85,B 0,C 180,E1 -28043.693,E2 -28043.693} C_VEL
LIN {X 0,Y 111.737,Z 519.435,A -85,B 0,C 180,E1 -28048.114,E2 -28048.114} C_VEL
LIN {X 0,Y 120.177,Z 510.053,A -85,B 0,C 180,E1 -28051.304,E2 -28051.304} C_VEL
LIN {X 0,Y 128.288,Z 499.387,A -85,B 0,C 180,E1 -28054.006,E2 -28054.006} C_VEL
LIN {X 0,Y 135.509,Z 488.201,A -85,B 0,C 180,E1 -28056.075,E2 -28056.075} C_VEL
LIN {X 0,Y 142.355,Z 475.484,A -85,B 0,C 180,E1 -28057.767,E2 -28057.767} C_VEL
LIN {X 0,Y 147.746,Z 463.098,A -85,B 0,C 180,E1 -28058.987,E2 -28058.987} C_VEL
LIN {X 0,Y 152.346,Z 449.604,A -85,B 0,C 180,E1 -28059.939,E2 -28059.939} C_VEL
LIN {X 0,Y 155.895,Z 435.104,A -85,B 0,C 180,E1 -28060.672,E2 -28060.672} C_VEL
LIN {X 0,Y 158.081,Z 420.806,A -85,B 0,C 180,E1 -28061.121,E2 -28061.121} C_VEL
LIN {X 0,Y 159.647,Z 406.219,A -85,B 0,C 180,E1 -28061.467,E2 -28061.467} C_VEL
LIN {X 0,Y 157.729,Z 401.227,A -85,B 0,C 180,E1 -28064.493,E2 -28064.493} C_VEL
LIN {X 0,Y 156.047,Z 397.351,A -85,B 0,C 180,E1 -28067.709,E2 -28067.709} C_VEL
LIN {X 0,Y 155.189,Z 395.323,A -85,B 0,C 180,E1 -28069.773,E2 -28069.773} C_VEL
LIN {X 0,Y 154.311,Z 393.024,A -85,B 0,C 180,E1 -28072.558,E2 -28072.558} C_VEL
LIN {X 0,Y 153.437,Z 389.682,A -85,B 0,C 180,E1 -28080,E2 -28080} C_VEL
LIN {X 0,Y 154.485,Z 393.381,A -85,B 0,C 180,E1 -28087.953,E2 -28087.953} C_VEL
LIN {X 0,Y 155.923,Z 397.057,A -85,B 0,C 180,E1 -28091.929,E2 -28091.929} C_VEL
LIN {X 0,Y 157.638,Z 401.026,A -85,B 0,C 180,E1 -28095.267,E2 -28095.267} C_VEL
LIN {X 0,Y 159.66,Z 406.219,A -85,B 0,C 180,E1 -28098.46,E2 -28098.46} C_VEL
LIN {X 0,Y 156.781,Z 430.716,A -85,B 0,C 180,E1 -28099.113,E2 -28099.113} C_VEL
LIN {X 0,Y 153.618,Z 445.533,A -85,B 0,C 180,E1 -28099.704,E2 -28099.704} C_VEL
LIN {X 0,Y 149.172,Z 459.852,A -85,B 0,C 180,E1 -28100.552,E2 -28100.552} C_VEL
LIN {X 0,Y 143.735,Z 473.21,A -85,B 0,C 180,E1 -28101.722,E2 -28101.722} C_VEL
LIN {X 0,Y 137.587,Z 485.272,A -85,B 0,C 180,E1 -28103.158,E2 -28103.158} C_VEL
LIN {X 0,Y 130.028,Z 497.451,A -85,B 0,C 180,E1 -28105.134,E2 -28105.134} C_VEL
LIN {X 0,Y 123.009,Z 507.183,A -85,B 0,C 180,E1 -28107.347,E2 -28107.347} C_VEL
LIN {X 0,Y 114.213,Z 517.527,A -85,B 0,C 180,E1 -28110.52,E2 -28110.52} C_VEL
LIN {X 0,Y 105.99,Z 525.838,A -85,B 0,C 180,E1 -28114.021,E2 -28114.021} C_VEL
LIN {X 0,Y 97.072,Z 533.787,A -85,B 0,C 180,E1 -28118.897,E2 -28118.897} C_VEL
LIN {X 0,Y 89.033,Z 540.187,A -85,B 0,C 180,E1 -28124.732,E2 -28124.732} C_VEL
LIN {X 0,Y 81.2,Z 545.862,A -85,B 0,C 180,E1 -28132.71,E2 -28132.71} C_VEL
LIN {X 0,Y 75.042,Z 549.978,A -85,B 0,C 180,E1 -28142.079,E2 -28142.079} C_VEL
LIN {X 0,Y 71.189,Z 552.667,A -85,B 0,C 180,E1 -28152.773,E2 -28152.773} C_VEL
LIN {X 0,Y 69.573,Z 553.995,A -85,B 0,C 180,E1 -28164.203,E2 -28164.203} C_VEL
LIN {X 0,Y 69.574,Z 554.156,A -85,B 0,C 180,E1 -28170,E2 -28170} C_VEL
LIN {X 0,Y 70.111,Z 553.469,A -85,B 0,C 180,E1 -28181.565,E2 -28181.565} C_VEL
LIN {X 0,Y 72.823,Z 551.44,A -85,B 0,C 180,E1 -28192.707,E2 -28192.707} C_VEL
LIN {X 0,Y 77.916,Z 548.021,A -85,B 0,C 180,E1 -28202.765,E2 -28202.765} C_VEL
LIN {X 0,Y 84.851,Z 543.109,A -85,B 0,C 180,E1 -28211.499,E2 -28211.499} C_VEL
LIN {X 0,Y 93.5,Z 536.561,A -85,B 0,C 180,E1 -28218.733,E2 -28218.733} C_VEL
LIN {X 0,Y 102.101,Z 529.278,A -85,B 0,C 180,E1 -28223.977,E2 -28223.977} C_VEL
LIN {X 0,Y 110.031,Z 521.643,A -85,B 0,C 180,E1 -28227.812,E2 -28227.812} C_VEL
LIN {X 0,Y 118.413,Z 512.485,A -85,B 0,C 180,E1 -28231.095,E2 -28231.095} C_VEL
LIN {X 0,Y 125.64,Z 503.351,A -85,B 0,C 180,E1 -28233.507,E2 -28233.507} C_VEL
LIN {X 0,Y 133.01,Z 492.452,A -85,B 0,C 180,E1 -28235.705,E2 -28235.705} C_VEL
LIN {X 0,Y 139.892,Z 480.518,A -85,B 0,C 180,E1 -28237.387,E2 -28237.387} C_VEL
LIN {X 0,Y 146.069,Z 467.279,A -85,B 0,C 180,E1 -28238.779,E2 -28238.779} C_VEL
LIN {X 0,Y 151.064,Z 453.479,A -85,B 0,C 180,E1 -28239.807,E2 -28239.807} C_VEL
LIN {X 0,Y 154.679,Z 440.028,A -85,B 0,C 180,E1 -28240.51,E2 -28240.51} C_VEL
LIN {X 0,Y 157.193,Z 426.017,A -85,B 0,C 180,E1 -28240.992,E2 -28240.992} C_VEL
LIN {X 0,Y 158.433,Z 414.951,A -85,B 0,C 180,E1 -28241.302,E2 -28241.302} C_VEL
LIN {X 0,Y 158.473,Z 412.61,A -85,B 0,C 180,E1 -28241.584,E2 -28241.584} C_VEL
LIN {X 0,Y 158.104,Z 410.223,A -85,B 0,C 180,E1 -28242.333,E2 -28242.333} C_VEL
LIN {X 0,Y 157.2,Z 407.91,A -85,B 0,C 180,E1 -28243.756,E2 -28243.756} C_VEL
LIN {X 0,Y 154.747,Z 404.422,A -85,B 0,C 180,E1 -28247.946,E2 -28247.946} C_VEL
LIN {X 0,Y 153.625,Z 401.526,A -85,B 0,C 180,E1 -28250.869,E2 -28250.869} C_VEL
LIN {X 0,Y 153.01,Z 399.702,A -85,B 0,C 180,E1 -28253.075,E2 -28253.075} C_VEL
LIN {X 0,Y 152.288,Z 396.256,A -85,B 0,C 180,E1 -28260,E2 -28260} C_VEL
LIN {X 0,Y 153.215,Z 400.312,A -85,B 0,C 180,E1 -28267.91,E2 -28267.91} C_VEL
LIN {X 0,Y 154.553,Z 403.92,A -85,B 0,C 180,E1 -28271.779,E2 -28271.779} C_VEL
LIN {X 0,Y 156.034,Z 407.655,A -85,B 0,C 180,E1 -28274.844,E2 -28274.844} C_VEL
LIN {X 0,Y 156.824,Z 409.84,A -85,B 0,C 180,E1 -28276.259,E2 -28276.259} C_VEL
LIN {X 0,Y 154.297,Z 430.262,A -85,B 0,C 180,E1 -28276.798,E2 -28276.798} C_VEL
LIN {X 0,Y 151.053,Z 445.057,A -85,B 0,C 180,E1 -28277.381,E2 -28277.381} C_VEL
LIN {X 0,Y 146.581,Z 459.177,A -85,B 0,C 180,E1 -28278.21,E2 -28278.21} C_VEL
LIN {X 0,Y 141.45,Z 471.594,A -85,B 0,C 180,E1 -28279.265,E2 -28279.265} C_VEL
LIN {X 0,Y 135.176,Z 483.778,A -85,B 0,C 180,E1 -28280.637,E2 -28280.637} C_VEL
LIN {X 0,Y 128.276,Z 494.898,A -85,B 0,C 180,E1 -28282.36,E2 -28282.36} C_VEL
LIN {X 0,Y 121.473,Z 504.261,A -85,B 0,C 180,E1 -28284.326,E2 -28284.326} C_VEL
LIN {X 0,Y 112.567,Z 514.68,A -85,B 0,C 180,E1 -28287.168,E2 -28287.168} C_VEL
LIN {X 0,Y 103.992,Z 523.272,A -85,B 0,C 180,E1 -28290.497,E2 -28290.497} C_VEL
LIN {X 0,Y 94.493,Z 531.504,A -85,B 0,C 180,E1 -28295.102,E2 -28295.102} C_VEL
LIN {X 0,Y 86.914,Z 537.246,A -85,B 0,C 180,E1 -28299.81,E2 -28299.81} C_VEL
LIN {X 0,Y 78.082,Z 543.355,A -85,B 0,C 180,E1 -28307.542,E2 -28307.542} C_VEL
LIN {X 0,Y 72.428,Z 546.84,A -85,B 0,C 180,E1 -28314.395,E2 -28314.395} C_VEL
LIN {X 0,Y 66.641,Z 550.233,A -85,B 0,C 180,E1 -28325.049,E2 -28325.049} C_VEL
LIN {X 0,Y 63.365,Z 552.24,A -85,B 0,C 180,E1 -28337.184,E2 -28337.184} C_VEL
LIN {X 0,Y 62.548,Z 552.917,A -85,B 0,C 180,E1 -28350,E2 -28350} C_VEL
LIN {X 0,Y 63.358,Z 552.281,A -85,B 0,C 180,E1 -28362.817,E2 -28362.817} C_VEL
LIN {X 0,Y 66.627,Z 550.31,A -85,B 0,C 180,E1 -28374.956,E2 -28374.956} C_VEL
LIN {X 0,Y 72.399,Z 546.955,A -85,B 0,C 180,E1 -28385.621,E2 -28385.621} C_VEL
LIN {X 0,Y 80.137,Z 542.117,A -85,B 0,C 180,E1 -28394.554,E2 -28394.554} C_VEL
LIN {X 0,Y 89.318,Z 535.641,A -85,B 0,C 180,E1 -28401.89,E2 -28401.89} C_VEL
LIN {X 0,Y 98.422,Z 528.427,A -85,B 0,C 180,E1 -28407.035,E2 -28407.035} C_VEL
LIN {X 0,Y 108.149,Z 519.5,A -85,B 0,C 180,E1 -28411.315,E2 -28411.315} C_VEL
LIN {X 0,Y 116.926,Z 510.117,A -85,B 0,C 180,E1 -28414.366,E2 -28414.366} C_VEL
LIN {X 0,Y 125.686,Z 498.96,A -85,B 0,C 180,E1 -28417.021,E2 -28417.021} C_VEL
LIN {X 0,Y 133.561,Z 486.973,A -85,B 0,C 180,E1 -28419.065,E2 -28419.065} C_VEL
LIN {X 0,Y 139.824,Z 475.545,A -85,B 0,C 180,E1 -28420.46,E2 -28420.46} C_VEL
LIN {X 0,Y 145.355,Z 463.158,A -85,B 0,C 180,E1 -28421.596,E2 -28421.596} C_VEL
LIN {X 0,Y 149.84,Z 450.387,A -85,B 0,C 180,E1 -28422.441,E2 -28422.441} C_VEL
LIN {X 0,Y 153.499,Z 436.07,A -85,B 0,C 180,E1 -28423.126,E2 -28423.126} C_VEL
LIN {X 0,Y 155.744,Z 422.32,A -85,B 0,C 180,E1 -28423.551,E2 -28423.551} C_VEL
LIN {X 0,Y 157.099,Z 410.054,A -85,B 0,C 180,E1 -28423.853,E2 -28423.853} C_VEL
LIN {X 0,Y 155.275,Z 405.267,A -85,B 0,C 180,E1 -28427.336,E2 -28427.336} C_VEL
LIN {X 0,Y 153.998,Z 402.019,A -85,B 0,C 180,E1 -28430.537,E2 -28430.537} C_VEL
LIN {X 0,Y 153.214,Z 399.83,A -85,B 0,C 180,E1 -28433.332,E2 -28433.332} C_VEL
LIN {X 0,Y 152.56,Z 396.822,A -85,B 0,C 180,E1 -28440,E2 -28440} C_VEL
LIN {X 0,Y 153.424,Z 400.317,A -85,B 0,C 180,E1 -28447.402,E2 -28447.402} C_VEL
LIN {X 0,Y 154.675,Z 403.757,A -85,B 0,C 180,E1 -28451.196,E2 -28451.196} C_VEL
LIN {X 0,Y 156.339,Z 407.954,A -85,B 0,C 180,E1 -28454.698,E2 -28454.698} C_VEL
LIN {X 0,Y 157.089,Z 410.116,A -85,B 0,C 180,E1 -28456.057,E2 -28456.057} C_VEL
LIN {X 0,Y 154.708,Z 430.079,A -85,B 0,C 180,E1 -28456.613,E2 -28456.613} C_VEL
LIN {X 0,Y 151.571,Z 444.754,A -85,B 0,C 180,E1 -28457.151,E2 -28457.151} C_VEL
LIN {X 0,Y 147.222,Z 458.663,A -85,B 0,C 180,E1 -28457.873,E2 -28457.873} C_VEL
LIN {X 0,Y 142.052,Z 471.384,A -85,B 0,C 180,E1 -28458.883,E2 -28458.883} C_VEL
LIN {X 0,Y 135.731,Z 483.792,A -85,B 0,C 180,E1 -28460.204,E2 -28460.204} C_VEL
LIN {X 0,Y 128.713,Z 495.138,A -85,B 0,C 180,E1 -28461.842,E2 -28461.842} C_VEL
LIN {X 0,Y 120.967,Z 505.767,A -85,B 0,C 180,E1 -28463.997,E2 -28463.997} C_VEL
LIN {X 0,Y 112.234,Z 515.953,A -85,B 0,C 180,E1 -28466.836,E2 -28466.836} C_VEL
LIN {X 0,Y 103.564,Z 524.517,A -85,B 0,C 180,E1 -28470.094,E2 -28470.094} C_VEL
LIN {X 0,Y 94.071,Z 532.713,A -85,B 0,C 180,E1 -28474.737,E2 -28474.737} C_VEL
LIN {X 0,Y 86.51,Z 538.461,A -85,B 0,C 180,E1 -28479.488,E2 -28479.488} C_VEL
LIN {X 0,Y 79.69,Z 543.164,A -85,B 0,C 180,E1 -28485.129,E2 -28485.129} C_VEL
LIN {X 0,Y 72.031,Z 548.04,A -85,B 0,C 180,E1 -28494.169,E2 -28494.169} C_VEL
LIN {X 0,Y 66.275,Z 551.429,A -85,B 0,C 180,E1 -28504.903,E2 -28504.903} C_VEL
LIN {X 0,Y 63.149,Z 553.433,A -85,B 0,C 180,E1 -28517.14,E2 -28517.14} C_VEL
LIN {X 0,Y 62.492,Z 554.09,A -85,B 0,C 180,E1 -28530,E2 -28530} C_VEL
LIN {X 0,Y 63.152,Z 553.402,A -85,B 0,C 180,E1 -28542.86,E2 -28542.86} C_VEL
LIN {X 0,Y 66.283,Z 551.372,A -85,B 0,C 180,E1 -28555.095,E2 -28555.095} C_VEL
LIN {X 0,Y 72.022,Z 547.954,A -85,B 0,C 180,E1 -28565.837,E2 -28565.837} C_VEL
LIN {X 0,Y 79.637,Z 543.041,A -85,B 0,C 180,E1 -28574.91,E2 -28574.91} C_VEL
LIN {X 0,Y 88.948,Z 536.493,A -85,B 0,C 180,E1 -28582.196,E2 -28582.196} C_VEL
LIN {X 0,Y 98.076,Z 529.209,A -85,B 0,C 180,E1 -28587.349,E2 -28587.349} C_VEL
LIN {X 0,Y 106.412,Z 521.574,A -85,B 0,C 180,E1 -28591.055,E2 -28591.055} C_VEL
LIN {X 0,Y 115.135,Z 512.416,A -85,B 0,C 180,E1 -28594.203,E2 -28594.203} C_VEL
LIN {X 0,Y 122.623,Z 503.281,A -85,B 0,C 180,E1 -28596.492,E2 -28596.492} C_VEL
LIN {X 0,Y 130.246,Z 492.382,A -85,B 0,C 180,E1 -28598.558,E2 -28598.558} C_VEL
LIN {X 0,Y 137.316,Z 480.447,A -85,B 0,C 180,E1 -28600.125,E2 -28600.125} C_VEL
LIN {X 0,Y 143.65,Z 467.207,A -85,B 0,C 180,E1 -28601.422,E2 -28601.422} C_VEL
LIN {X 0,Y 148.652,Z 453.77,A -85,B 0,C 180,E1 -28602.351,E2 -28602.351} C_VEL
LIN {X 0,Y 152.445,Z 440.016,A -85,B 0,C 180,E1 -28603.02,E2 -28603.02} C_VEL
LIN {X 0,Y 155.075,Z 425.583,A -85,B 0,C 180,E1 -28603.479,E2 -28603.479} C_VEL
LIN {X 0,Y 156.799,Z 409.83,A -85,B 0,C 180,E1 -28603.951,E2 -28603.951} C_VEL
LIN {X 0,Y 155.155,Z 405.338,A -85,B 0,C 180,E1 -28607.079,E2 -28607.079} C_VEL
LIN {X 0,Y 154.747,Z 404.422,A -85,B 0,C 180,E1 -28607.946,E2 -28607.946} C_VEL
LIN {X 0,Y 154.1,Z 403.49,A -85,B 0,C 180,E1 -28609.346,E2 -28609.346} C_VEL
LIN {X 0,Y 153.151,Z 403.125,A -85,B 0,C 180,E1 -28611.527,E2 -28611.527} C_VEL
LIN {X 0,Y 151.584,Z 404.067,A -85,B 0,C 180,E1 -28616.761,E2 -28616.761} C_VEL
LIN {X 0,Y 151.384,Z 403.832,A -85,B 0,C 180,E1 -28619.026,E2 -28619.026} C_VEL
LIN {X 0,Y 151.4,Z 403.506,A -85,B 0,C 180,E1 -28619.773,E2 -28619.773} C_VEL
LIN {X 0,Y 151.372,Z 404.158,A -85,B 0,C 180,E1 -28621.621,E2 -28621.621} C_VEL
LIN {X 0,Y 152.16,Z 407.21,A -85,B 0,C 180,E1 -28627.339,E2 -28627.339} C_VEL
LIN {X 0,Y 153.179,Z 410.263,A -85,B 0,C 180,E1 -28630.682,E2 -28630.682} C_VEL
LIN {X 0,Y 154.531,Z 414.066,A -85,B 0,C 180,E1 -28633.841,E2 -28633.841} C_VEL
LIN {X 0,Y 152.158,Z 431.712,A -85,B 0,C 180,E1 -28634.293,E2 -28634.293} C_VEL
LIN {X 0,Y 148.86,Z 445.97,A -85,B 0,C 180,E1 -28634.811,E2 -28634.811} C_VEL
LIN {X 0,Y 144.523,Z 459.251,A -85,B 0,C 180,E1 -28635.54,E2 -28635.54} C_VEL
LIN {X 0,Y 139.273,Z 471.667,A -85,B 0,C 180,E1 -28636.512,E2 -28636.512} C_VEL
LIN {X 0,Y 132.836,Z 483.849,A -85,B 0,C 180,E1 -28637.765,E2 -28637.765} C_VEL
LIN {X 0,Y 125.134,Z 495.846,A -85,B 0,C 180,E1 -28639.509,E2 -28639.509} C_VEL
LIN {X 0,Y 117.186,Z 506.241,A -85,B 0,C 180,E1 -28641.633,E2 -28641.633} C_VEL
LIN {X 0,Y 107.979,Z 516.281,A -85,B 0,C 180,E1 -28644.329,E2 -28644.329} C_VEL
LIN {X 0,Y 99.111,Z 524.616,A -85,B 0,C 180,E1 -28647.581,E2 -28647.581} C_VEL
LIN {X 0,Y 89.201,Z 532.578,A -85,B 0,C 180,E1 -28652.117,E2 -28652.117} C_VEL
LIN {X 0,Y 80.001,Z 538.984,A -85,B 0,C 180,E1 -28657.756,E2 -28657.756} C_VEL
LIN {X 0,Y 70.816,Z 544.661,A -85,B 0,C 180,E1 -28665.997,E2 -28665.997} C_VEL
LIN {X 0,Y 63.151,Z 548.784,A -85,B 0,C 180,E1 -28676.19,E2 -28676.19} C_VEL
LIN {X 0,Y 58.014,Z 551.472,A -85,B 0,C 180,E1 -28688.689,E2 -28688.689} C_VEL
LIN {X 0,Y 55.564,Z 552.811,A -85,B 0,C 180,E1 -28702.733,E2 -28702.733} C_VEL
LIN {X 0,Y 55.466,Z 552.984,A -85,B 0,C 180,E1 -28710,E2 -28710} C_VEL
LIN {X 0,Y 56.452,Z 552.347,A -85,B 0,C 180,E1 -28724.417,E2 -28724.417} C_VEL
LIN {X 0,Y 60.25,Z 550.376,A -85,B 0,C 180,E1 -28737.812,E2 -28737.812} C_VEL
LIN {X 0,Y 66.724,Z 547.021,A -85,B 0,C 180,E1 -28749.195,E2 -28749.195} C_VEL
LIN {X 0,Y 75.223,Z 542.182,A -85,B 0,C 180,E1 -28758.366,E2 -28758.366} C_VEL
LIN {X 0,Y 85.108,Z 535.707,A -85,B 0,C 180,E1 -28765.664,E2 -28765.664} C_VEL
LIN {X 0,Y 94.736,Z 528.492,A -85,B 0,C 180,E1 -28770.651,E2 -28770.651} C_VEL
LIN {X 0,Y 104.911,Z 519.564,A -85,B 0,C 180,E1 -28774.734,E2 -28774.734} C_VEL
LIN {X 0,Y 114.027,Z 510.181,A -85,B 0,C 180,E1 -28777.591,E2 -28777.591} C_VEL
LIN {X 0,Y 122.994,Z 499.152,A -85,B 0,C 180,E1 -28780.042,E2 -28780.042} C_VEL
LIN {X 0,Y 131.185,Z 487.036,A -85,B 0,C 180,E1 -28781.971,E2 -28781.971} C_VEL
LIN {X 0,Y 137.615,Z 475.607,A -85,B 0,C 180,E1 -28783.243,E2 -28783.243} C_VEL
LIN {X 0,Y 143.276,Z 463.218,A -85,B 0,C 180,E1 -28784.285,E2 -28784.285} C_VEL
LIN {X 0,Y 148.089,Z 449.688,A -85,B 0,C 180,E1 -28785.106,E2 -28785.106} C_VEL
LIN {X 0,Y 151.772,Z 435.318,A -85,B 0,C 180,E1 -28785.722,E2 -28785.722} C_VEL
LIN {X 0,Y 154.111,Z 420.624,A -85,B 0,C 180,E1 -28786.118,E2 -28786.118} C_VEL
LIN {X 0,Y 154.812,Z 414.247,A -85,B 0,C 180,E1 -28786.276,E2 -28786.276} C_VEL
LIN {X 0,Y 153.275,Z 409.944,A -85,B 0,C 180,E1 -28789.962,E2 -28789.962} C_VEL
LIN {X 0,Y 152.168,Z 406.63,A -85,B 0,C 180,E1 -28794.035,E2 -28794.035} C_VEL
LIN {X 0,Y 151.683,Z 403.961,A -85,B 0,C 180,E1 -28800,E2 -28800} C_VEL
LIN {X 0,Y 152.363,Z 407.126,A -85,B 0,C 180,E1 -28806.746,E2 -28806.746} C_VEL
LIN {X 0,Y 153.432,Z 410.448,A -85,B 0,C 180,E1 -28810.407,E2 -28810.407} C_VEL
LIN {X 0,Y 154.796,Z 414.259,A -85,B 0,C 180,E1 -28813.615,E2 -28813.615} C_VEL
LIN {X 0,Y 154.291,Z 419.276,A -85,B 0,C 180,E1 -28813.81,E2 -28813.81} C_VEL
LIN {X 0,Y 152.041,Z 434.431,A -85,B 0,C 180,E1 -28814.19,E2 -28814.19} C_VEL
LIN {X 0,Y 148.547,Z 448.679,A -85,B 0,C 180,E1 -28814.73,E2 -28814.73} C_VEL
LIN {X 0,Y 143.986,Z 461.886,A -85,B 0,C 180,E1 -28815.425,E2 -28815.425} C_VEL
LIN {X 0,Y 138.299,Z 474.709,A -85,B 0,C 180,E1 -28816.432,E2 -28816.432} C_VEL
LIN {X 0,Y 131.832,Z 486.453,A -85,B 0,C 180,E1 -28817.656,E2 -28817.656} C_VEL
LIN {X 0,Y 124.65,Z 497.325,A -85,B 0,C 180,E1 -28819.2,E2 -28819.2} C_VEL
LIN {X 0,Y 116.057,Z 508.32,A -85,B 0,C 180,E1 -28821.456,E2 -28821.456} C_VEL
LIN {X 0,Y 107.676,Z 517.398,A -85,B 0,C 180,E1 -28823.971,E2 -28823.971} C_VEL
LIN {X 0,Y 98.728,Z 525.709,A -85,B 0,C 180,E1 -28827.153,E2 -28827.153} C_VEL
LIN {X 0,Y 88.81,Z 533.656,A -85,B 0,C 180,E1 -28831.714,E2 -28831.714} C_VEL
LIN {X 0,Y 79.611,Z 540.056,A -85,B 0,C 180,E1 -28837.393,E2 -28837.393} C_VEL
LIN {X 0,Y 70.382,Z 545.731,A -85,B 0,C 180,E1 -28845.656,E2 -28845.656} C_VEL
LIN {X 0,Y 62.806,Z 549.846,A -85,B 0,C 180,E1 -28855.98,E2 -28855.98} C_VEL
LIN {X 0,Y 57.712,Z 552.534,A -85,B 0,C 180,E1 -28868.573,E2 -28868.573} C_VEL
LIN {X 0,Y 55.46,Z 553.862,A -85,B 0,C 180,E1 -28882.72,E2 -28882.72} C_VEL
LIN {X 0,Y 55.393,Z 554.023,A -85,B 0,C 180,E1 -28890,E2 -28890} C_VEL
LIN {X 0,Y 56.243,Z 553.335,A -85,B 0,C 180,E1 -28904.473,E2 -28904.473} C_VEL
LIN {X 0,Y 59.885,Z 551.305,A -85,B 0,C 180,E1 -28917.997,E2 -28917.997} C_VEL
LIN {X 0,Y 66.354,Z 547.886,A -85,B 0,C 180,E1 -28929.456,E2 -28929.456} C_VEL
LIN {X 0,Y 74.828,Z 542.907,A -85,B 0,C 180,E1 -28938.894,E2 -28938.894} C_VEL
LIN {X 0,Y 84.765,Z 536.425,A -85,B 0,C 180,E1 -28946.007,E2 -28946.007} C_VEL
LIN {X 0,Y 94.404,Z 529.14,A -85,B 0,C 180,E1 -28951.012,E2 -28951.012} C_VEL
LIN {X 0,Y 103.155,Z 521.505,A -85,B 0,C 180,E1 -28954.517,E2 -28954.517} C_VEL
LIN {X 0,Y 112.221,Z 512.346,A -85,B 0,C 180,E1 -28957.476,E2 -28957.476} C_VEL
LIN {X 0,Y 121.515,Z 501.227,A -85,B 0,C 180,E1 -28960.022,E2 -28960.022} C_VEL
LIN {X 0,Y 129.423,Z 489.874,A -85,B 0,C 180,E1 -28961.856,E2 -28961.856} C_VEL
LIN {X 0,Y 136.678,Z 477.316,A -85,B 0,C 180,E1 -28963.273,E2 -28963.273} C_VEL
LIN {X 0,Y 142.356,Z 465.15,A -85,B 0,C 180,E1 -28964.298,E2 -28964.298} C_VEL
LIN {X 0,Y 147.428,Z 451.22,A -85,B 0,C 180,E1 -28965.13,E2 -28965.13} C_VEL
LIN {X 0,Y 151.183,Z 436.997,A -85,B 0,C 180,E1 -28965.711,E2 -28965.711} C_VEL
LIN {X 0,Y 153.595,Z 422.654,A -85,B 0,C 180,E1 -28966.086,E2 -28966.086} C_VEL
LIN {X 0,Y 154.521,Z 413.996,A -85,B 0,C 180,E1 -28966.365,E2 -28966.365} C_VEL
LIN {X 0,Y 152.872,Z 409.23,A -85,B 0,C 180,E1 -28970.407,E2 -28970.407} C_VEL
LIN {X 0,Y 151.933,Z 406.452,A -85,B 0,C 180,E1 -28973.86,E2 -28973.86} C_VEL
LIN {X 0,Y 151.4,Z 403.506,A -85,B 0,C 180,E1 -28979.773,E2 -28979.773} C_VEL
LIN {X 0,Y 151.437,Z 403.425,A -85,B 0,C 180,E1 -28981.216,E2 -28981.216} C_VEL
LIN {X 0,Y 151.432,Z 404.789,A -85,B 0,C 180,E1 -28982.972,E2 -28982.972} C_VEL
LIN {X 0,Y 151.42,Z 408.304,A -85,B 0,C 180,E1 -28985.238,E2 -28985.238} C_VEL
LIN {X 0,Y 151.777,Z 415.768,A -85,B 0,C 180,E1 -28989.129,E2 -28989.129} C_VEL
LIN {X 0,Y 152.186,Z 417.649,A -85,B 0,C 180,E1 -28990.54,E2 -28990.54} C_VEL
LIN {X 0,Y 152.476,Z 418.483,A -85,B 0,C 180,E1 -28991.314,E2 -28991.314} C_VEL
LIN {X 0,Y 150.331,Z 433.086,A -85,B 0,C 180,E1 -28991.717,E2 -28991.717} C_VEL
LIN {X 0,Y 147.077,Z 446.508,A -85,B 0,C 180,E1 -28992.152,E2 -28992.152} C_VEL
LIN {X 0,Y 142.378,Z 460.436,A -85,B 0,C 180,E1 -28992.871,E2 -28992.871} C_VEL
LIN {X 0,Y 136.592,Z 473.428,A -85,B 0,C 180,E1 -28993.798,E2 -28993.798} C_VEL
LIN {X 0,Y 129.211,Z 486.557,A -85,B 0,C 180,E1 -28995.108,E2 -28995.108} C_VEL
LIN {X 0,Y 121.273,Z 498.136,A -85,B 0,C 180,E1 -28996.755,E2 -28996.755} C_VEL
LIN {X 0,Y 113.17,Z 508.089,A -85,B 0,C 180,E1 -28998.733,E2 -28998.733} C_VEL
LIN {X 0,Y 103.68,Z 517.833,A -85,B 0,C 180,E1 -29001.245,E2 -29001.245} C_VEL
LIN {X 0,Y 94.507,Z 525.914,A -85,B 0,C 180,E1 -29004.362,E2 -29004.362} C_VEL
LIN {X 0,Y 84.187,Z 533.652,A -85,B 0,C 180,E1 -29008.773,E2 -29008.773} C_VEL
LIN {X 0,Y 73.995,Z 540.172,A -85,B 0,C 180,E1 -29014.742,E2 -29014.742} C_VEL
LIN {X 0,Y 65.858,Z 544.729,A -85,B 0,C 180,E1 -29021.67,E2 -29021.67} C_VEL
LIN {X 0,Y 57.362,Z 548.851,A -85,B 0,C 180,E1 -29032.223,E2 -29032.223} C_VEL
LIN {X 0,Y 51.443,Z 551.539,A -85,B 0,C 180,E1 -29045.805,E2 -29045.805} C_VEL
LIN {X 0,Y 48.525,Z 552.878,A -85,B 0,C 180,E1 -29061.672,E2 -29061.672} C_VEL
LIN {X 0,Y 48.368,Z 553.05,A -85,B 0,C 180,E1 -29069.999,E2 -29069.999} C_VEL
LIN {X 0,Y 49.587,Z 552.414,A -85,B 0,C 180,E1 -29086.466,E2 -29086.466} C_VEL
LIN {X 0,Y 54.044,Z 550.442,A -85,B 0,C 180,E1 -29101.342,E2 -29101.342} C_VEL
LIN {X 0,Y 61.362,Z 547.087,A -85,B 0,C 180,E1 -29113.407,E2 -29113.407} C_VEL
LIN {X 0,Y 70.689,Z 542.248,A -85,B 0,C 180,E1 -29122.688,E2 -29122.688} C_VEL
LIN {X 0,Y 81.302,Z 535.772,A -85,B 0,C 180,E1 -29129.815,E2 -29129.815} C_VEL
LIN {X 0,Y 91.451,Z 528.557,A -85,B 0,C 180,E1 -29134.549,E2 -29134.549} C_VEL
LIN {X 0,Y 102.077,Z 519.629,A -85,B 0,C 180,E1 -29138.349,E2 -29138.349} C_VEL
LIN {X 0,Y 111.509,Z 510.245,A -85,B 0,C 180,E1 -29140.973,E2 -29140.973} C_VEL
LIN {X 0,Y 120.746,Z 499.215,A -85,B 0,C 180,E1 -29143.224,E2 -29143.224} C_VEL
LIN {X 0,Y 129.165,Z 487.098,A -85,B 0,C 180,E1 -29144.965,E2 -29144.965} C_VEL
LIN {X 0,Y 135.738,Z 475.668,A -85,B 0,C 180,E1 -29146.114,E2 -29146.114} C_VEL
LIN {X 0,Y 141.516,Z 463.278,A -85,B 0,C 180,E1 -29147.058,E2 -29147.058} C_VEL
LIN {X 0,Y 146.526,Z 449.433,A -85,B 0,C 180,E1 -29147.805,E2 -29147.805} C_VEL
LIN {X 0,Y 150.271,Z 434.961,A -85,B 0,C 180,E1 -29148.365,E2 -29148.365} C_VEL
LIN {X 0,Y 152.657,Z 419.872,A -85,B 0,C 180,E1 -29148.718,E2 -29148.718} C_VEL
LIN {X 0,Y 152.738,Z 418.647,A -85,B 0,C 180,E1 -29148.856,E2 -29148.856} C_VEL
LIN {X 0,Y 151.726,Z 415.476,A -85,B 0,C 180,E1 -29152.012,E2 -29152.012} C_VEL
LIN {X 0,Y 151.16,Z 413.471,A -85,B 0,C 180,E1 -29154.664,E2 -29154.664} C_VEL
LIN {X 0,Y 150.809,Z 411.085,A -85,B 0,C 180,E1 -29160,E2 -29160} C_VEL
LIN {X 0,Y 151.338,Z 414.005,A -85,B 0,C 180,E1 -29166.165,E2 -29166.165} C_VEL
LIN {X 0,Y 152.226,Z 417.143,A -85,B 0,C 180,E1 -29169.623,E2 -29169.623} C_VEL
LIN {X 0,Y 152.787,Z 418.784,A -85,B 0,C 180,E1 -29171.184,E2 -29171.184} C_VEL
LIN {X 0,Y 150.462,Z 434.383,A -85,B 0,C 180,E1 -29171.575,E2 -29171.575} C_VEL
LIN {X 0,Y 147.36,Z 447.004,A -85,B 0,C 180,E1 -29171.982,E2 -29171.982} C_VEL
LIN {X 0,Y 142.674,Z 460.798,A -85,B 0,C 180,E1 -29172.6,E2 -29172.6} C_VEL
LIN {X 0,Y 137.284,Z 473.027,A -85,B 0,C 180,E1 -29173.433,E2 -29173.433} C_VEL
LIN {X 0,Y 130.679,Z 485.085,A -85,B 0,C 180,E1 -29174.528,E2 -29174.528} C_VEL
LIN {X 0,Y 122.497,Z 497.261,A -85,B 0,C 180,E1 -29176.06,E2 -29176.06} C_VEL
LIN {X 0,Y 114.783,Z 506.979,A -85,B 0,C 180,E1 -29177.827,E2 -29177.827} C_VEL
LIN {X 0,Y 104.983,Z 517.333,A -85,B 0,C 180,E1 -29180.414,E2 -29180.414} C_VEL
LIN {X 0,Y 95.677,Z 525.644,A -85,B 0,C 180,E1 -29183.341,E2 -29183.341} C_VEL
LIN {X 0,Y 85.278,Z 533.591,A -85,B 0,C 180,E1 -29187.636,E2 -29187.636} C_VEL
LIN {X 0,Y 75.486,Z 539.99,A -85,B 0,C 180,E1 -29193.081,E2 -29193.081} C_VEL
LIN {X 0,Y 65.468,Z 545.665,A -85,B 0,C 180,E1 -29201.286,E2 -29201.286} C_VEL
LIN {X 0,Y 57.045,Z 549.78,A -85,B 0,C 180,E1 -29211.977,E2 -29211.977} C_VEL
LIN {X 0,Y 51.125,Z 552.468,A -85,B 0,C 180,E1 -29225.645,E2 -29225.645} C_VEL
LIN {X 0,Y 48.412,Z 553.795,A -85,B 0,C 180,E1 -29241.654,E2 -29241.654} C_VEL
LIN {X 0,Y 48.309,Z 553.957,A -85,B 0,C 180,E1 -29250.001,E2 -29250.001} C_VEL
LIN {X 0,Y 49.367,Z 553.268,A -85,B 0,C 180,E1 -29266.542,E2 -29266.542} C_VEL
LIN {X 0,Y 53.68,Z 551.237,A -85,B 0,C 180,E1 -29281.58,E2 -29281.58} C_VEL
LIN {X 0,Y 60.991,Z 547.818,A -85,B 0,C 180,E1 -29293.739,E2 -29293.739} C_VEL
LIN {X 0,Y 70.229,Z 542.904,A -85,B 0,C 180,E1 -29303.184,E2 -29303.184} C_VEL
LIN {X 0,Y 80.982,Z 536.356,A -85,B 0,C 180,E1 -29310.207,E2 -29310.207} C_VEL
LIN {X 0,Y 91.155,Z 529.071,A -85,B 0,C 180,E1 -29314.945,E2 -29314.945} C_VEL
LIN {X 0,Y 101.847,Z 520.043,A -85,B 0,C 180,E1 -29318.679,E2 -29318.679} C_VEL
LIN {X 0,Y 111.293,Z 510.574,A -85,B 0,C 180,E1 -29321.3,E2 -29321.3} C_VEL
LIN {X 0,Y 120.065,Z 500.087,A -85,B 0,C 180,E1 -29323.434,E2 -29323.434} C_VEL
LIN {X 0,Y 127.394,Z 489.804,A -85,B 0,C 180,E1 -29324.887,E2 -29324.887} C_VEL
LIN {X 0,Y 134.804,Z 477.245,A -85,B 0,C 180,E1 -29326.166,E2 -29326.166} C_VEL
LIN {X 0,Y 140.604,Z 465.077,A -85,B 0,C 180,E1 -29327.079,E2 -29327.079} C_VEL
LIN {X 0,Y 145.503,Z 451.976,A -85,B 0,C 180,E1 -29327.789,E2 -29327.789} C_VEL
LIN {X 0,Y 149.338,Z 438.013,A -85,B 0,C 180,E1 -29328.316,E2 -29328.316} C_VEL
LIN {X 0,Y 151.951,Z 423.228,A -85,B 0,C 180,E1 -29328.674,E2 -29328.674} C_VEL
LIN {X 0,Y 152.48,Z 418.441,A -85,B 0,C 180,E1 -29328.865,E2 -29328.865} C_VEL
LIN {X 0,Y 151.33,Z 414.862,A -85,B 0,C 180,E1 -29332.495,E2 -29332.495} C_VEL
LIN {X 0,Y 150.885,Z 413.199,A -85,B 0,C 180,E1 -29334.655,E2 -29334.655} C_VEL
LIN {X 0,Y 150.53,Z 410.577,A -85,B 0,C 180,E1 -29340,E2 -29340} C_VEL
LIN {X 0,Y 151.12,Z 414.106,A -85,B 0,C 180,E1 -29346.761,E2 -29346.761} C_VEL
LIN {X 0,Y 152.047,Z 417.181,A -85,B 0,C 180,E1 -29350.129,E2 -29350.129} C_VEL
LIN {X 0,Y 152.186,Z 417.649,A -85,B 0,C 180,E1 -29350.54,E2 -29350.54} C_VEL
LIN {X 0,Y 152.249,Z 419.013,A -85,B 0,C 180,E1 -29351,E2 -29351} C_VEL
LIN {X 0,Y 152.001,Z 421.534,A -85,B 0,C 180,E1 -29351.145,E2 -29351.145} C_VEL
LIN {X 0,Y 151.317,Z 425.18,A -85,B 0,C 180,E1 -29350.837,E2 -29350.837} C_VEL
LIN {X 0,Y 148.926,Z 434.352,A -85,B 0,C 180,E1 -29349.304,E2 -29349.304} C_VEL
LIN {X 0,Y 147.942,Z 438.207,A -85,B 0,C 180,E1 -29349.162,E2 -29349.162} C_VEL
LIN {X 0,Y 143.922,Z 452.375,A -85,B 0,C 180,E1 -29349.662,E2 -29349.662} C_VEL
LIN {X 0,Y 138.437,Z 466.483,A -85,B 0,C 180,E1 -29350.395,E2 -29350.395} C_VEL
LIN {X 0,Y 131.724,Z 479.72,A -85,B 0,C 180,E1 -29351.373,E2 -29351.373} C_VEL
LIN {X 0,Y 124.211,Z 491.643,A -85,B 0,C 180,E1 -29352.577,E2 -29352.577} C_VEL
LIN {X 0,Y 115.969,Z 502.523,A -85,B 0,C 180,E1 -29354.16,E2 -29354.16} C_VEL
LIN {X 0,Y 107.818,Z 511.639,A -85,B 0,C 180,E1 -29355.962,E2 -29355.962} C_VEL
LIN {X 0,Y 98.114,Z 520.777,A -85,B 0,C 180,E1 -29358.36,E2 -29358.36} C_VEL
LIN {X 0,Y 87.12,Z 529.502,A -85,B 0,C 180,E1 -29361.922,E2 -29361.922} C_VEL
LIN {X 0,Y 77.998,Z 535.647,A -85,B 0,C 180,E1 -29365.705,E2 -29365.705} C_VEL
LIN {X 0,Y 69.474,Z 540.639,A -85,B 0,C 180,E1 -29370.385,E2 -29370.385} C_VEL
LIN {X 0,Y 61.338,Z 544.797,A -85,B 0,C 180,E1 -29376.675,E2 -29376.675} C_VEL
LIN {X 0,Y 51.912,Z 548.919,A -85,B 0,C 180,E1 -29387.398,E2 -29387.398} C_VEL
LIN {X 0,Y 45.048,Z 551.607,A -85,B 0,C 180,E1 -29402.093,E2 -29402.093} C_VEL
LIN {X 0,Y 41.501,Z 552.945,A -85,B 0,C 180,E1 -29420.25,E2 -29420.25} C_VEL
LIN {X 0,Y 41.285,Z 553.117,A -85,B 0,C 180,E1 -29429.999,E2 -29429.999} C_VEL
LIN {X 0,Y 42.816,Z 552.48,A -85,B 0,C 180,E1 -29449.164,E2 -29449.164} C_VEL
LIN {X 0,Y 48.085,Z 550.508,A -85,B 0,C 180,E1 -29465.775,E2 -29465.775} C_VEL
LIN {X 0,Y 56.397,Z 547.153,A -85,B 0,C 180,E1 -29478.39,E2 -29478.39} C_VEL
LIN {X 0,Y 66.599,Z 542.314,A -85,B 0,C 180,E1 -29487.585,E2 -29487.585} C_VEL
LIN {X 0,Y 77.96,Z 535.837,A -85,B 0,C 180,E1 -29494.351,E2 -29494.351} C_VEL
LIN {X 0,Y 88.621,Z 528.622,A -85,B 0,C 180,E1 -29498.716,E2 -29498.716} C_VEL
LIN {X 0,Y 99.675,Z 519.693,A -85,B 0,C 180,E1 -29502.148,E2 -29502.148} C_VEL
LIN {X 0,Y 109.398,Z 510.309,A -85,B 0,C 180,E1 -29504.496,E2 -29504.496} C_VEL
LIN {X 0,Y 118.392,Z 499.923,A -85,B 0,C 180,E1 -29506.409,E2 -29506.409} C_VEL
LIN {X 0,Y 126.673,Z 488.451,A -85,B 0,C 180,E1 -29507.915,E2 -29507.915} C_VEL
LIN {X 0,Y 134.21,Z 475.73,A -85,B 0,C 180,E1 -29509.061,E2 -29509.061} C_VEL
LIN {X 0,Y 140.098,Z 463.338,A -85,B 0,C 180,E1 -29509.886,E2 -29509.886} C_VEL
LIN {X 0,Y 144.911,Z 450.366,A -85,B 0,C 180,E1 -29510.5,E2 -29510.5} C_VEL
LIN {X 0,Y 148.725,Z 436.235,A -85,B 0,C 180,E1 -29510.992,E2 -29510.992} C_VEL
LIN {X 0,Y 150.932,Z 423.533,A -85,B 0,C 180,E1 -29511.347,E2 -29511.347} C_VEL
LIN {X 0,Y 150.205,Z 420.42,A -85,B 0,C 180,E1 -29515.085,E2 -29515.085} C_VEL
LIN {X 0,Y 149.923,Z 418.313,A -85,B 0,C 180,E1 -29520.21,E2 -29520.21} C_VEL
LIN {X 0,Y 150.329,Z 420.87,A -85,B 0,C 180,E1 -29525.575,E2 -29525.575} C_VEL
LIN {X 0,Y 150.961,Z 423.605,A -85,B 0,C 180,E1 -29528.641,E2 -29528.641} C_VEL
LIN {X 0,Y 148.395,Z 437.915,A -85,B 0,C 180,E1 -29528.986,E2 -29528.986} C_VEL
LIN {X 0,Y 144.455,Z 452.007,A -85,B 0,C 180,E1 -29529.432,E2 -29529.432} C_VEL
LIN {X 0,Y 140.029,Z 463.753,A -85,B 0,C 180,E1 -29529.954,E2 -29529.954} C_VEL
LIN {X 0,Y 134.127,Z 476.168,A -85,B 0,C 180,E1 -29530.753,E2 -29530.753} C_VEL
LIN {X 0,Y 126.562,Z 488.913,A -85,B 0,C 180,E1 -29531.85,E2 -29531.85} C_VEL
LIN {X 0,Y 118.235,Z 500.408,A -85,B 0,C 180,E1 -29533.264,E2 -29533.264} C_VEL
LIN {X 0,Y 109.221,Z 510.828,A -85,B 0,C 180,E1 -29535.166,E2 -29535.166} C_VEL
LIN {X 0,Y 99.49,Z 520.241,A -85,B 0,C 180,E1 -29537.518,E2 -29537.518} C_VEL
LIN {X 0,Y 89.931,Z 528.044,A -85,B 0,C 180,E1 -29540.322,E2 -29540.322} C_VEL
LIN {X 0,Y 80.687,Z 534.535,A -85,B 0,C 180,E1 -29543.859,E2 -29543.859} C_VEL
LIN {X 0,Y 71.834,Z 539.924,A -85,B 0,C 180,E1 -29548.296,E2 -29548.296} C_VEL
LIN {X 0,Y 60.994,Z 545.599,A -85,B 0,C 180,E1 -29556.24,E2 -29556.24} C_VEL
LIN {X 0,Y 51.603,Z 549.714,A -85,B 0,C 180,E1 -29567.082,E2 -29567.082} C_VEL
LIN {X 0,Y 44.72,Z 552.401,A -85,B 0,C 180,E1 -29581.872,E2 -29581.872} C_VEL
LIN {X 0,Y 41.397,Z 553.729,A -85,B 0,C 180,E1 -29600.226,E2 -29600.226} C_VEL
LIN {X 0,Y 41.198,Z 553.89,A -85,B 0,C 180,E1 -29610.001,E2 -29610.001} C_VEL
LIN {X 0,Y 42.586,Z 553.201,A -85,B 0,C 180,E1 -29629.273,E2 -29629.273} C_VEL
LIN {X 0,Y 47.741,Z 551.17,A -85,B 0,C 180,E1 -29646.075,E2 -29646.075} C_VEL
LIN {X 0,Y 56.036,Z 547.75,A -85,B 0,C 180,E1 -29658.808,E2 -29658.808} C_VEL
LIN {X 0,Y 66.198,Z 542.836,A -85,B 0,C 180,E1 -29668.137,E2 -29668.137} C_VEL
LIN {X 0,Y 77.681,Z 536.288,A -85,B 0,C 180,E1 -29674.784,E2 -29674.784} C_VEL
LIN {X 0,Y 88.369,Z 529.003,A -85,B 0,C 180,E1 -29679.142,E2 -29679.142} C_VEL
LIN {X 0,Y 99.483,Z 519.974,A -85,B 0,C 180,E1 -29682.496,E2 -29682.496} C_VEL
LIN {X 0,Y 109.224,Z 510.505,A -85,B 0,C 180,E1 -29684.83,E2 -29684.83} C_VEL
LIN {X 0,Y 118.229,Z 500.017,A -85,B 0,C 180,E1 -29686.749,E2 -29686.749} C_VEL
LIN {X 0,Y 126.568,Z 488.441,A -85,B 0,C 180,E1 -29688.14,E2 -29688.14} C_VEL
LIN {X 0,Y 134.133,Z 475.591,A -85,B 0,C 180,E1 -29689.235,E2 -29689.235} C_VEL
LIN {X 0,Y 140.039,Z 463.015,A -85,B 0,C 180,E1 -29690.024,E2 -29690.024} C_VEL
LIN {X 0,Y 144.598,Z 450.581,A -85,B 0,C 180,E1 -29690.6,E2 -29690.6} C_VEL
LIN {X 0,Y 148.305,Z 436.903,A -85,B 0,C 180,E1 -29691.028,E2 -29691.028} C_VEL
LIN {X 0,Y 150.671,Z 423.355,A -85,B 0,C 180,E1 -29691.358,E2 -29691.358} C_VEL
LIN {X 0,Y 149.948,Z 420.203,A -85,B 0,C 180,E1 -29694.959,E2 -29694.959} C_VEL
LIN {X 0,Y 149.648,Z 417.761,A -85,B 0,C 180,E1 -29700,E2 -29700} C_VEL
LIN {X 0,Y 150.076,Z 420.877,A -85,B 0,C 180,E1 -29706.049,E2 -29706.049} C_VEL
LIN {X 0,Y 150.651,Z 423.28,A -85,B 0,C 180,E1 -29708.767,E2 -29708.767} C_VEL
LIN {X 0,Y 148.732,Z 434.814,A -85,B 0,C 180,E1 -29709.081,E2 -29709.081} C_VEL
LIN {X 0,Y 147.942,Z 438.207,A -85,B 0,C 180,E1 -29709.162,E2 -29709.162} C_VEL
LIN {X 0,Y 146.975,Z 442.027,A -85,B 0,C 180,E1 -29709.171,E2 -29709.171} C_VEL
LIN {X 0,Y 144.579,Z 449.475,A -85,B 0,C 180,E1 -29708.693,E2 -29708.693} C_VEL
LIN {X 0,Y 139.418,Z 462.048,A -85,B 0,C 180,E1 -29707.535,E2 -29707.535} C_VEL
LIN {X 0,Y 136.932,Z 467.401,A -85,B 0,C 180,E1 -29707.529,E2 -29707.529} C_VEL
LIN {X 0,Y 130.509,Z 479.791,A -85,B 0,C 180,E1 -29708.315,E2 -29708.315} C_VEL
LIN {X 0,Y 122.861,Z 491.713,A -85,B 0,C 180,E1 -29709.345,E2 -29709.345} C_VEL
LIN {X 0,Y 113.662,Z 503.492,A -85,B 0,C 180,E1 -29710.837,E2 -29710.837} C_VEL
LIN {X 0,Y 104.412,Z 513.333,A -85,B 0,C 180,E1 -29712.584,E2 -29712.584} C_VEL
LIN {X 0,Y 94.457,Z 522.197,A -85,B 0,C 180,E1 -29714.706,E2 -29714.706} C_VEL
LIN {X 0,Y 84.724,Z 529.571,A -85,B 0,C 180,E1 -29717.46,E2 -29717.46} C_VEL
LIN {X 0,Y 75.181,Z 535.715,A -85,B 0,C 180,E1 -29720.805,E2 -29720.805} C_VEL
LIN {X 0,Y 65.435,Z 541.073,A -85,B 0,C 180,E1 -29725.444,E2 -29725.444} C_VEL
LIN {X 0,Y 54.64,Z 546.05,A -85,B 0,C 180,E1 -29733.276,E2 -29733.276} C_VEL
LIN {X 0,Y 46.918,Z 548.986,A -85,B 0,C 180,E1 -29741.5,E2 -29741.5} C_VEL
LIN {X 0,Y 38.894,Z 551.674,A -85,B 0,C 180,E1 -29757.174,E2 -29757.174} C_VEL
LIN {X 0,Y 34.525,Z 553.011,A -85,B 0,C 180,E1 -29778.254,E2 -29778.254} C_VEL
LIN {X 0,Y 34.175,Z 553.183,A -85,B 0,C 180,E1 -29789.999,E2 -29789.999} C_VEL
LIN {X 0,Y 36.184,Z 552.547,A -85,B 0,C 180,E1 -29812.857,E2 -29812.857} C_VEL
LIN {X 0,Y 42.495,Z 550.575,A -85,B 0,C 180,E1 -29831.416,E2 -29831.416} C_VEL
LIN {X 0,Y 51.94,Z 547.219,A -85,B 0,C 180,E1 -29844.275,E2 -29844.275} C_VEL
LIN {X 0,Y 63.059,Z 542.38,A -85,B 0,C 180,E1 -29853.072,E2 -29853.072} C_VEL
LIN {X 0,Y 72.05,Z 537.707,A -85,B 0,C 180,E1 -29857.916,E2 -29857.916} C_VEL
LIN {X 0,Y 83.074,Z 530.914,A -85,B 0,C 180,E1 -29862.123,E2 -29862.123} C_VEL
LIN {X 0,Y 92.791,Z 523.827,A -85,B 0,C 180,E1 -29864.94,E2 -29864.94} C_VEL
LIN {X 0,Y 102.714,Z 515.29,A -85,B 0,C 180,E1 -29867.161,E2 -29867.161} C_VEL
LIN {X 0,Y 112.199,Z 505.542,A -85,B 0,C 180,E1 -29869.02,E2 -29869.02} C_VEL
LIN {X 0,Y 121.146,Z 494.537,A -85,B 0,C 180,E1 -29870.467,E2 -29870.467} C_VEL
LIN {X 0,Y 128.788,Z 483.216,A -85,B 0,C 180,E1 -29871.516,E2 -29871.516} C_VEL
LIN {X 0,Y 135.611,Z 470.834,A -85,B 0,C 180,E1 -29872.36,E2 -29872.36} C_VEL
LIN {X 0,Y 141.59,Z 457.012,A -85,B 0,C 180,E1 -29873.074,E2 -29873.074} C_VEL
LIN {X 0,Y 146.088,Z 443.154,A -85,B 0,C 180,E1 -29873.507,E2 -29873.507} C_VEL
LIN {X 0,Y 149.292,Z 428.562,A -85,B 0,C 180,E1 -29873.939,E2 -29873.939} C_VEL
LIN {X 0,Y 149.07,Z 427.138,A -85,B 0,C 180,E1 -29875.962,E2 -29875.962} C_VEL
LIN {X 0,Y 148.966,Z 425.382,A -85,B 0,C 180,E1 -29880,E2 -29880} C_VEL
LIN {X 0,Y 149.192,Z 427.653,A -85,B 0,C 180,E1 -29884.898,E2 -29884.898} C_VEL
LIN {X 0,Y 149.321,Z 428.625,A -85,B 0,C 180,E1 -29886.049,E2 -29886.049} C_VEL
LIN {X 0,Y 146.301,Z 442.568,A -85,B 0,C 180,E1 -29886.377,E2 -29886.377} C_VEL
LIN {X 0,Y 142.143,Z 455.758,A -85,B 0,C 180,E1 -29886.763,E2 -29886.763} C_VEL
LIN {X 0,Y 137.268,Z 467.609,A -85,B 0,C 180,E1 -29887.272,E2 -29887.272} C_VEL
LIN {X 0,Y 130.419,Z 480.69,A -85,B 0,C 180,E1 -29888.043,E2 -29888.043} C_VEL
LIN {X 0,Y 122.738,Z 492.537,A -85,B 0,C 180,E1 -29888.992,E2 -29888.992} C_VEL
LIN {X 0,Y 114.283,Z 503.364,A -85,B 0,C 180,E1 -29890.291,E2 -29890.291} C_VEL
LIN {X 0,Y 104.224,Z 514.068,A -85,B 0,C 180,E1 -29892.114,E2 -29892.114} C_VEL
LIN {X 0,Y 94.27,Z 522.904,A -85,B 0,C 180,E1 -29894.27,E2 -29894.27} C_VEL
LIN {X 0,Y 84.481,Z 530.256,A -85,B 0,C 180,E1 -29896.929,E2 -29896.929} C_VEL
LIN {X 0,Y 74.924,Z 536.385,A -85,B 0,C 180,E1 -29900.284,E2 -29900.284} C_VEL
LIN {X 0,Y 62.769,Z 542.9,A -85,B 0,C 180,E1 -29906.401,E2 -29906.401} C_VEL
LIN {X 0,Y 51.624,Z 547.775,A -85,B 0,C 180,E1 -29915.234,E2 -29915.234} C_VEL
LIN {X 0,Y 42.173,Z 551.163,A -85,B 0,C 180,E1 -29928.198,E2 -29928.198} C_VEL
LIN {X 0,Y 35.943,Z 553.167,A -85,B 0,C 180,E1 -29946.981,E2 -29946.981} C_VEL
LIN {X 0,Y 34.092,Z 553.824,A -85,B 0,C 180,E1 -29970.001,E2 -29970.001} C_VEL
LIN {X 0,Y 35.946,Z 553.134,A -85,B 0,C 180,E1 -29993.019,E2 -29993.019} C_VEL
LIN {X 0,Y 42.176,Z 551.102,A -85,B 0,C 180,E1 -30011.8,E2 -30011.8} C_VEL
LIN {X 0,Y 51.604,Z 547.682,A -85,B 0,C 180,E1 -30024.799,E2 -30024.799} C_VEL
LIN {X 0,Y 62.72,Z 542.768,A -85,B 0,C 180,E1 -30033.691,E2 -30033.691} C_VEL
LIN {X 0,Y 74.923,Z 536.219,A -85,B 0,C 180,E1 -30039.721,E2 -30039.721} C_VEL
LIN {X 0,Y 86.08,Z 528.934,A -85,B 0,C 180,E1 -30043.599,E2 -30043.599} C_VEL
LIN {X 0,Y 97.581,Z 519.905,A -85,B 0,C 180,E1 -30046.479,E2 -30046.479} C_VEL
LIN {X 0,Y 108.245,Z 509.728,A -85,B 0,C 180,E1 -30048.615,E2 -30048.615} C_VEL
LIN {X 0,Y 117.65,Z 498.876,A -85,B 0,C 180,E1 -30050.278,E2 -30050.278} C_VEL
LIN {X 0,Y 126.153,Z 487.079,A -85,B 0,C 180,E1 -30051.431,E2 -30051.431} C_VEL
LIN {X 0,Y 132.99,Z 475.519,A -85,B 0,C 180,E1 -30052.241,E2 -30052.241} C_VEL
LIN {X 0,Y 139.413,Z 461.948,A -85,B 0,C 180,E1 -30052.957,E2 -30052.957} C_VEL
LIN {X 0,Y 144.384,Z 448.137,A -85,B 0,C 180,E1 -30053.48,E2 -30053.48} C_VEL
LIN {X 0,Y 147.978,Z 434.064,A -85,B 0,C 180,E1 -30053.802,E2 -30053.802} C_VEL
LIN {X 0,Y 149.037,Z 428.322,A -85,B 0,C 180,E1 -30053.977,E2 -30053.977} C_VEL
LIN {X 0,Y 148.788,Z 426.844,A -85,B 0,C 180,E1 -30056.022,E2 -30056.022} C_VEL
LIN {X 0,Y 148.687,Z 424.951,A -85,B 0,C 180,E1 -30060,E2 -30060} C_VEL
LIN {X 0,Y 148.929,Z 427.67,A -85,B 0,C 180,E1 -30065.416,E2 -30065.416} C_VEL
LIN {X 0,Y 149.025,Z 428.336,A -85,B 0,C 180,E1 -30066.226,E2 -30066.226} C_VEL
LIN {X 0,Y 145.812,Z 442.942,A -85,B 0,C 180,E1 -30066.572,E2 -30066.572} C_VEL
LIN {X 0,Y 141.614,Z 456.085,A -85,B 0,C 180,E1 -30067.003,E2 -30067.003} C_VEL
LIN {X 0,Y 136.932,Z 467.401,A -85,B 0,C 180,E1 -30067.529,E2 -30067.529} C_VEL
LIN {X 0,Y 134.264,Z 472.749,A -85,B 0,C 180,E1 -30067.553,E2 -30067.553} C_VEL
LIN {X 0,Y 129.22,Z 481.185,A -85,B 0,C 180,E1 -30066.844,E2 -30066.844} C_VEL
LIN {X 0,Y 123.75,Z 489.265,A -85,B 0,C 180,E1 -30066.142,E2 -30066.142} C_VEL
LIN {X 0,Y 120.306,Z 493.966,A -85,B 0,C 180,E1 -30066.233,E2 -30066.233} C_VEL
LIN {X 0,Y 111.981,Z 504.2,A -85,B 0,C 180,E1 -30067.358,E2 -30067.358} C_VEL
LIN {X 0,Y 103.099,Z 513.402,A -85,B 0,C 180,E1 -30068.73,E2 -30068.73} C_VEL
LIN {X 0,Y 92.906,Z 522.266,A -85,B 0,C 180,E1 -30070.458,E2 -30070.458} C_VEL
LIN {X 0,Y 81.199,Z 530.753,A -85,B 0,C 180,E1 -30073.169,E2 -30073.169} C_VEL
LIN {X 0,Y 69.698,Z 537.587,A -85,B 0,C 180,E1 -30076.681,E2 -30076.681} C_VEL
LIN {X 0,Y 60.163,Z 542.299,A -85,B 0,C 180,E1 -30080.85,E2 -30080.85} C_VEL
LIN {X 0,Y 48.157,Z 547.178,A -85,B 0,C 180,E1 -30088.881,E2 -30088.881} C_VEL
LIN {X 0,Y 37.451,Z 550.571,A -85,B 0,C 180,E1 -30101.354,E2 -30101.354} C_VEL
LIN {X 0,Y 29.752,Z 552.575,A -85,B 0,C 180,E1 -30121.807,E2 -30121.807} C_VEL
LIN {X 0,Y 27.07,Z 553.25,A -85,B 0,C 180,E1 -30149.999,E2 -30149.999} C_VEL
LIN {X 0,Y 29.747,Z 552.613,A -85,B 0,C 180,E1 -30178.196,E2 -30178.196} C_VEL
LIN {X 0,Y 37.438,Z 550.641,A -85,B 0,C 180,E1 -30198.665,E2 -30198.665} C_VEL
LIN {X 0,Y 48.132,Z 547.285,A -85,B 0,C 180,E1 -30211.172,E2 -30211.172} C_VEL
LIN {X 0,Y 60.165,Z 542.445,A -85,B 0,C 180,E1 -30219.143,E2 -30219.143} C_VEL
LIN {X 0,Y 69.684,Z 537.773,A -85,B 0,C 180,E1 -30223.355,E2 -30223.355} C_VEL
LIN {X 0,Y 81.174,Z 530.979,A -85,B 0,C 180,E1 -30226.903,E2 -30226.903} C_VEL
LIN {X 0,Y 91.201,Z 523.891,A -85,B 0,C 180,E1 -30229.263,E2 -30229.263} C_VEL
LIN {X 0,Y 101.372,Z 515.354,A -85,B 0,C 180,E1 -30231.082,E2 -30231.082} C_VEL
LIN {X 0,Y 110.461,Z 506.275,A -85,B 0,C 180,E1 -30232.54,E2 -30232.54} C_VEL
LIN {X 0,Y 119.314,Z 495.763,A -85,B 0,C 180,E1 -30233.702,E2 -30233.702} C_VEL
LIN {X 0,Y 127.067,Z 484.692,A -85,B 0,C 180,E1 -30234.587,E2 -30234.587} C_VEL
LIN {X 0,Y 133.986,Z 472.657,A -85,B 0,C 180,E1 -30235.262,E2 -30235.262} C_VEL
LIN {X 0,Y 140.047,Z 459.329,A -85,B 0,C 180,E1 -30235.842,E2 -30235.842} C_VEL
LIN {X 0,Y 144.762,Z 445.64,A -85,B 0,C 180,E1 -30236.24,E2 -30236.24} C_VEL
LIN {X 0,Y 147.697,Z 433.955,A -85,B 0,C 180,E1 -30236.548,E2 -30236.548} C_VEL
LIN {X 0,Y 147.732,Z 432.448,A -85,B 0,C 180,E1 -30240,E2 -30240} C_VEL
LIN {X 0,Y 147.726,Z 433.876,A -85,B 0,C 180,E1 -30243.384,E2 -30243.384} C_VEL
LIN {X 0,Y 144.082,Z 448.094,A -85,B 0,C 180,E1 -30243.718,E2 -30243.718} C_VEL
LIN {X 0,Y 139.152,Z 461.645,A -85,B 0,C 180,E1 -30244.08,E2 -30244.08} C_VEL
LIN {X 0,Y 133.082,Z 474.462,A -85,B 0,C 180,E1 -30244.619,E2 -30244.619} C_VEL
LIN {X 0,Y 126.157,Z 486.204,A -85,B 0,C 180,E1 -30245.276,E2 -30245.276} C_VEL
LIN {X 0,Y 117.522,Z 498.141,A -85,B 0,C 180,E1 -30246.187,E2 -30246.187} C_VEL
LIN {X 0,Y 108.034,Z 508.976,A -85,B 0,C 180,E1 -30247.475,E2 -30247.475} C_VEL
LIN {X 0,Y 97.867,Z 518.628,A -85,B 0,C 180,E1 -30249.111,E2 -30249.111} C_VEL
LIN {X 0,Y 87.705,Z 526.682,A -85,B 0,C 180,E1 -30251.009,E2 -30251.009} C_VEL
LIN {X 0,Y 76.044,Z 534.405,A -85,B 0,C 180,E1 -30253.98,E2 -30253.98} C_VEL
LIN {X 0,Y 66.266,Z 539.793,A -85,B 0,C 180,E1 -30257.354,E2 -30257.354} C_VEL
LIN {X 0,Y 53.782,Z 545.466,A -85,B 0,C 180,E1 -30263.837,E2 -30263.837} C_VEL
LIN {X 0,Y 42.277,Z 549.581,A -85,B 0,C 180,E1 -30273.782,E2 -30273.782} C_VEL
LIN {X 0,Y 32.83,Z 552.268,A -85,B 0,C 180,E1 -30290.045,E2 -30290.045} C_VEL
LIN {X 0,Y 27.485,Z 553.596,A -85,B 0,C 180,E1 -30315.186,E2 -30315.186} C_VEL
LIN {X 0,Y 27,Z 553.757,A -85,B 0,C 180,E1 -30330.001,E2 -30330.001} C_VEL
LIN {X 0,Y 29.509,Z 553.067,A -85,B 0,C 180,E1 -30358.446,E2 -30358.446} C_VEL
LIN {X 0,Y 37.156,Z 551.035,A -85,B 0,C 180,E1 -30379.164,E2 -30379.164} C_VEL
LIN {X 0,Y 47.841,Z 547.614,A -85,B 0,C 180,E1 -30391.813,E2 -30391.813} C_VEL
LIN {X 0,Y 59.901,Z 542.7,A -85,B 0,C 180,E1 -30399.818,E2 -30399.818} C_VEL
LIN {X 0,Y 72.755,Z 536.151,A -85,B 0,C 180,E1 -30405.008,E2 -30405.008} C_VEL
LIN {X 0,Y 84.343,Z 528.865,A -85,B 0,C 180,E1 -30408.255,E2 -30408.255} C_VEL
LIN {X 0,Y 96.168,Z 519.836,A -85,B 0,C 180,E1 -30410.6,E2 -30410.6} C_VEL
LIN {X 0,Y 106.39,Z 510.365,A -85,B 0,C 180,E1 -30412.251,E2 -30412.251} C_VEL
LIN {X 0,Y 115.798,Z 499.876,A -85,B 0,C 180,E1 -30413.621,E2 -30413.621} C_VEL
LIN {X 0,Y 124.427,Z 488.3,A -85,B 0,C 180,E1 -30414.557,E2 -30414.557} C_VEL
LIN {X 0,Y 132.219,Z 475.448,A -85,B 0,C 180,E1 -30415.291,E2 -30415.291} C_VEL
LIN {X 0,Y 138.722,Z 461.875,A -85,B 0,C 180,E1 -30415.867,E2 -30415.867} C_VEL
LIN {X 0,Y 143.787,Z 447.948,A -85,B 0,C 180,E1 -30416.292,E2 -30416.292} C_VEL
LIN {X 0,Y 147.429,Z 433.675,A -85,B 0,C 180,E1 -30416.613,E2 -30416.613} C_VEL
LIN {X 0,Y 147.462,Z 432.069,A -85,B 0,C 180,E1 -30420,E2 -30420} C_VEL
LIN {X 0,Y 147.407,Z 433.722,A -85,B 0,C 180,E1 -30423.553,E2 -30423.553} C_VEL
LIN {X 0,Y 144.237,Z 446.285,A -85,B 0,C 180,E1 -30423.85,E2 -30423.85} C_VEL
LIN {X 0,Y 139.624,Z 459.546,A -85,B 0,C 180,E1 -30424.254,E2 -30424.254} C_VEL
LIN {X 0,Y 134,Z 471.955,A -85,B 0,C 180,E1 -30424.803,E2 -30424.803} C_VEL
LIN {X 0,Y 127.082,Z 484.134,A -85,B 0,C 180,E1 -30425.479,E2 -30425.479} C_VEL
LIN {X 0,Y 120.306,Z 493.966,A -85,B 0,C 180,E1 -30426.233,E2 -30426.233} C_VEL
LIN {X 0,Y 116.669,Z 498.632,A -85,B 0,C 180,E1 -30426.367,E2 -30426.367} C_VEL
LIN {X 0,Y 110.101,Z 505.981,A -85,B 0,C 180,E1 -30425.739,E2 -30425.739} C_VEL
LIN {X 0,Y 103.047,Z 512.855,A -85,B 0,C 180,E1 -30425.06,E2 -30425.06} C_VEL
LIN {X 0,Y 98.623,Z 516.776,A -85,B 0,C 180,E1 -30425.221,E2 -30425.221} C_VEL
LIN {X 0,Y 88.443,Z 524.96,A -85,B 0,C 180,E1 -30426.648,E2 -30426.648} C_VEL
LIN {X 0,Y 76.472,Z 532.92,A -85,B 0,C 180,E1 -30428.906,E2 -30428.906} C_VEL
LIN {X 0,Y 64.636,Z 539.325,A -85,B 0,C 180,E1 -30431.881,E2 -30431.881} C_VEL
LIN {X 0,Y 51.498,Z 545,A -85,B 0,C 180,E1 -30437.198,E2 -30437.198} C_VEL
LIN {X 0,Y 38.975,Z 549.121,A -85,B 0,C 180,E1 -30445.633,E2 -30445.633} C_VEL
LIN {X 0,Y 27.987,Z 551.809,A -85,B 0,C 180,E1 -30461.12,E2 -30461.12} C_VEL
LIN {X 0,Y 20.829,Z 553.145,A -85,B 0,C 180,E1 -30490.279,E2 -30490.279} C_VEL
LIN {X 0,Y 19.98,Z 553.316,A -85,B 0,C 180,E1 -30509.999,E2 -30509.999} C_VEL
LIN {X 0,Y 23.714,Z 552.68,A -85,B 0,C 180,E1 -30546.348,E2 -30546.348} C_VEL
LIN {X 0,Y 33.159,Z 550.708,A -85,B 0,C 180,E1 -30567.969,E2 -30567.969} C_VEL
LIN {X 0,Y 45.131,Z 547.351,A -85,B 0,C 180,E1 -30579.116,E2 -30579.116} C_VEL
LIN {X 0,Y 58.003,Z 542.511,A -85,B 0,C 180,E1 -30585.768,E2 -30585.768} C_VEL
LIN {X 0,Y 67.986,Z 537.838,A -85,B 0,C 180,E1 -30589.122,E2 -30589.122} C_VEL
LIN {X 0,Y 79.864,Z 531.044,A -85,B 0,C 180,E1 -30591.879,E2 -30591.879} C_VEL
LIN {X 0,Y 91.869,Z 522.605,A -85,B 0,C 180,E1 -30593.976,E2 -30593.976} C_VEL
LIN {X 0,Y 102.249,Z 513.795,A -85,B 0,C 180,E1 -30595.29,E2 -30595.29} C_VEL
LIN {X 0,Y 112.651,Z 503.12,A -85,B 0,C 180,E1 -30596.532,E2 -30596.532} C_VEL
LIN {X 0,Y 121.359,Z 492.318,A -85,B 0,C 180,E1 -30597.359,E2 -30597.359} C_VEL
LIN {X 0,Y 129.217,Z 480.491,A -85,B 0,C 180,E1 -30597.97,E2 -30597.97} C_VEL
LIN {X 0,Y 136.211,Z 467.429,A -85,B 0,C 180,E1 -30598.495,E2 -30598.495} C_VEL
LIN {X 0,Y 141.667,Z 454.327,A -85,B 0,C 180,E1 -30598.863,E2 -30598.863} C_VEL
LIN {X 0,Y 146.083,Z 439.827,A -85,B 0,C 180,E1 -30599.182,E2 -30599.182} C_VEL
LIN {X 0,Y 146.154,Z 439.483,A -85,B 0,C 180,E1 -30600,E2 -30600} C_VEL
LIN {X 0,Y 146.098,Z 439.774,A -85,B 0,C 180,E1 -30600.685,E2 -30600.685} C_VEL
LIN {X 0,Y 142.626,Z 451.524,A -85,B 0,C 180,E1 -30600.961,E2 -30600.961} C_VEL
LIN {X 0,Y 137.952,Z 463.572,A -85,B 0,C 180,E1 -30601.215,E2 -30601.215} C_VEL
LIN {X 0,Y 131.824,Z 475.983,A -85,B 0,C 180,E1 -30601.616,E2 -30601.616} C_VEL
LIN {X 0,Y 123.954,Z 488.725,A -85,B 0,C 180,E1 -30602.169,E2 -30602.169} C_VEL
LIN {X 0,Y 115.226,Z 500.218,A -85,B 0,C 180,E1 -30602.876,E2 -30602.876} C_VEL
LIN {X 0,Y 105.663,Z 510.636,A -85,B 0,C 180,E1 -30603.91,E2 -30603.91} C_VEL
LIN {X 0,Y 95.266,Z 520.048,A -85,B 0,C 180,E1 -30605.189,E2 -30605.189} C_VEL
LIN {X 0,Y 84.905,Z 527.849,A -85,B 0,C 180,E1 -30606.651,E2 -30606.651} C_VEL
LIN {X 0,Y 74.643,Z 534.339,A -85,B 0,C 180,E1 -30608.662,E2 -30608.662} C_VEL
LIN {X 0,Y 64.499,Z 539.727,A -85,B 0,C 180,E1 -30611.295,E2 -30611.295} C_VEL
LIN {X 0,Y 51.31,Z 545.4,A -85,B 0,C 180,E1 -30616.512,E2 -30616.512} C_VEL
LIN {X 0,Y 38.766,Z 549.515,A -85,B 0,C 180,E1 -30624.983,E2 -30624.983} C_VEL
LIN {X 0,Y 27.742,Z 552.202,A -85,B 0,C 180,E1 -30640.539,E2 -30640.539} C_VEL
LIN {X 0,Y 20.681,Z 553.529,A -85,B 0,C 180,E1 -30670.135,E2 -30670.135} C_VEL
LIN {X 0,Y 19.897,Z 553.69,A -85,B 0,C 180,E1 -30690.001,E2 -30690.001} C_VEL
LIN {X 0,Y 23.489,Z 553,A -85,B 0,C 180,E1 -30726.757,E2 -30726.757} C_VEL
LIN {X 0,Y 32.934,Z 550.967,A -85,B 0,C 180,E1 -30748.603,E2 -30748.603} C_VEL
LIN {X 0,Y 44.91,Z 547.546,A -85,B 0,C 180,E1 -30759.871,E2 -30759.871} C_VEL
LIN {X 0,Y 57.825,Z 542.632,A -85,B 0,C 180,E1 -30766.482,E2 -30766.482} C_VEL
LIN {X 0,Y 71.244,Z 536.083,A -85,B 0,C 180,E1 -30770.556,E2 -30770.556} C_VEL
LIN {X 0,Y 83.186,Z 528.797,A -85,B 0,C 180,E1 -30773.069,E2 -30773.069} C_VEL
LIN {X 0,Y 95.264,Z 519.766,A -85,B 0,C 180,E1 -30774.828,E2 -30774.828} C_VEL
LIN {X 0,Y 105.664,Z 510.296,A -85,B 0,C 180,E1 -30776.09,E2 -30776.09} C_VEL
LIN {X 0,Y 115.225,Z 499.806,A -85,B 0,C 180,E1 -30777.137,E2 -30777.137} C_VEL
LIN {X 0,Y 123.955,Z 488.229,A -85,B 0,C 180,E1 -30777.827,E2 -30777.827} C_VEL
LIN {X 0,Y 131.825,Z 475.376,A -85,B 0,C 180,E1 -30778.376,E2 -30778.376} C_VEL
LIN {X 0,Y 137.954,Z 462.797,A -85,B 0,C 180,E1 -30778.768,E2 -30778.768} C_VEL
LIN {X 0,Y 143.22,Z 448.739,A -85,B 0,C 180,E1 -30779.104,E2 -30779.104} C_VEL
LIN {X 0,Y 145.838,Z 439.438,A -85,B 0,C 180,E1 -30779.272,E2 -30779.272} C_VEL
LIN {X 0,Y 145.9,Z 439.109,A -85,B 0,C 180,E1 -30780,E2 -30780} C_VEL
LIN {X 0,Y 145.823,Z 439.478,A -85,B 0,C 180,E1 -30780.887,E2 -30780.887} C_VEL
LIN {X 0,Y 141.391,Z 454.133,A -85,B 0,C 180,E1 -30781.196,E2 -30781.196} C_VEL
LIN {X 0,Y 136.214,Z 466.701,A -85,B 0,C 180,E1 -30781.546,E2 -30781.546} C_VEL
LIN {X 0,Y 129.222,Z 479.933,A -85,B 0,C 180,E1 -30782.084,E2 -30782.084} C_VEL
LIN {X 0,Y 121.366,Z 491.854,A -85,B 0,C 180,E1 -30782.711,E2 -30782.711} C_VEL
LIN {X 0,Y 112.665,Z 502.732,A -85,B 0,C 180,E1 -30783.577,E2 -30783.577} C_VEL
LIN {X 0,Y 103.996,Z 511.846,A -85,B 0,C 180,E1 -30784.596,E2 -30784.596} C_VEL
LIN {X 0,Y 98.623,Z 516.776,A -85,B 0,C 180,E1 -30785.221,E2 -30785.221} C_VEL
LIN {X 0,Y 94.057,Z 520.591,A -85,B 0,C 180,E1 -30785.409,E2 -30785.409} C_VEL
LIN {X 0,Y 86.123,Z 526.399,A -85,B 0,C 180,E1 -30784.647,E2 -30784.647} C_VEL
LIN {X 0,Y 77.867,Z 531.743,A -85,B 0,C 180,E1 -30783.772,E2 -30783.772} C_VEL
LIN {X 0,Y 72.766,Z 534.653,A -85,B 0,C 180,E1 -30783.989,E2 -30783.989} C_VEL
LIN {X 0,Y 59.762,Z 541.153,A -85,B 0,C 180,E1 -30786.435,E2 -30786.435} C_VEL
LIN {X 0,Y 46.473,Z 546.253,A -85,B 0,C 180,E1 -30790.593,E2 -30790.593} C_VEL
LIN {X 0,Y 36.468,Z 549.188,A -85,B 0,C 180,E1 -30795.512,E2 -30795.512} C_VEL
LIN {X 0,Y 23.911,Z 551.876,A -85,B 0,C 180,E1 -30808.144,E2 -30808.144} C_VEL
LIN {X 0,Y 14.349,Z 553.211,A -85,B 0,C 180,E1 -30840.672,E2 -30840.672} C_VEL
LIN {X 0,Y 12.878,Z 553.383,A -85,B 0,C 180,E1 -30869.998,E2 -30869.998} C_VEL
LIN {X 0,Y 18.476,Z 552.746,A -85,B 0,C 180,E1 -30919.53,E2 -30919.53} C_VEL
LIN {X 0,Y 29.991,Z 550.774,A -85,B 0,C 180,E1 -30939.607,E2 -30939.607} C_VEL
LIN {X 0,Y 43.105,Z 547.417,A -85,B 0,C 180,E1 -30948.023,E2 -30948.023} C_VEL
LIN {X 0,Y 56.671,Z 542.577,A -85,B 0,C 180,E1 -30952.785,E2 -30952.785} C_VEL
LIN {X 0,Y 67.006,Z 537.904,A -85,B 0,C 180,E1 -30955.128,E2 -30955.128} C_VEL
LIN {X 0,Y 79.171,Z 531.109,A -85,B 0,C 180,E1 -30957,E2 -30957} C_VEL
LIN {X 0,Y 91.397,Z 522.67,A -85,B 0,C 180,E1 -30958.408,E2 -30958.408} C_VEL
LIN {X 0,Y 102.993,Z 512.857,A -85,B 0,C 180,E1 -30959.371,E2 -30959.371} C_VEL
LIN {X 0,Y 105.42,Z 510.564,A -85,B 0,C 180,E1 -30959.571,E2 -30959.571} C_VEL
LIN {X 0,Y 105.772,Z 510.211,A -85,B 0,C 180,E1 -30960,E2 -30960} C_VEL
LIN {X 0,Y 94.887,Z 519.983,A -85,B 0,C 180,E1 -30960.9,E2 -30960.9} C_VEL
LIN {X 0,Y 82.629,Z 528.943,A -85,B 0,C 180,E1 -30962.047,E2 -30962.047} C_VEL
LIN {X 0,Y 70.426,Z 536.189,A -85,B 0,C 180,E1 -30963.721,E2 -30963.721} C_VEL
LIN {X 0,Y 60.033,Z 541.269,A -85,B 0,C 180,E1 -30965.7,E2 -30965.7} C_VEL
LIN {X 0,Y 46.365,Z 546.51,A -85,B 0,C 180,E1 -30969.856,E2 -30969.856} C_VEL
LIN {X 0,Y 36.334,Z 549.449,A -85,B 0,C 180,E1 -30974.737,E2 -30974.737} C_VEL
LIN {X 0,Y 23.724,Z 552.135,A -85,B 0,C 180,E1 -30987.292,E2 -30987.292} C_VEL
LIN {X 0,Y 14.2,Z 553.462,A -85,B 0,C 180,E1 -31020.338,E2 -31020.338} C_VEL
LIN {X 0,Y 12.786,Z 553.624,A -85,B 0,C 180,E1 -31050.002,E2 -31050.002} C_VEL
LIN {X 0,Y 18.288,Z 552.933,A -85,B 0,C 180,E1 -31100.227,E2 -31100.227} C_VEL
LIN {X 0,Y 29.846,Z 550.9,A -85,B 0,C 180,E1 -31120.374,E2 -31120.374} C_VEL
LIN {X 0,Y 42.98,Z 547.478,A -85,B 0,C 180,E1 -31128.843,E2 -31128.843} C_VEL
LIN {X 0,Y 56.584,Z 542.564,A -85,B 0,C 180,E1 -31133.525,E2 -31133.525} C_VEL
LIN {X 0,Y 70.427,Z 536.014,A -85,B 0,C 180,E1 -31136.283,E2 -31136.283} C_VEL
LIN {X 0,Y 82.628,Z 528.728,A -85,B 0,C 180,E1 -31137.995,E2 -31137.995} C_VEL
LIN {X 0,Y 94.888,Z 519.697,A -85,B 0,C 180,E1 -31139.113,E2 -31139.113} C_VEL
LIN {X 0,Y 105.773,Z 509.865,A -85,B 0,C 180,E1 -31140,E2 -31140} C_VEL
LIN {X 0,Y 105.423,Z 510.216,A -85,B 0,C 180,E1 -31140.539,E2 -31140.539} C_VEL
LIN {X 0,Y 94.903,Z 519.661,A -85,B 0,C 180,E1 -31141.367,E2 -31141.367} C_VEL
LIN {X 0,Y 84.412,Z 527.486,A -85,B 0,C 180,E1 -31142.458,E2 -31142.458} C_VEL
LIN {X 0,Y 72.766,Z 534.653,A -85,B 0,C 180,E1 -31143.989,E2 -31143.989} C_VEL
LIN {X 0,Y 66.998,Z 537.71,A -85,B 0,C 180,E1 -31144.365,E2 -31144.365} C_VEL
LIN {X 0,Y 57.068,Z 542.196,A -85,B 0,C 180,E1 -31143.524,E2 -31143.524} C_VEL
LIN {X 0,Y 48.924,Z 545.267,A -85,B 0,C 180,E1 -31142.509,E2 -31142.509} C_VEL
LIN {X 0,Y 42.699,Z 547.233,A -85,B 0,C 180,E1 -31142.512,E2 -31142.512} C_VEL
LIN {X 0,Y 40.617,Z 547.809,A -85,B 0,C 180,E1 -31142.867,E2 -31142.867} C_VEL
LIN {X 0,Y 28.309,Z 550.773,A -85,B 0,C 180,E1 -31146.772,E2 -31146.772} C_VEL
LIN {X 0,Y 14.874,Z 552.776,A -85,B 0,C 180,E1 -31159.091,E2 -31159.091} C_VEL
LIN {X 0,Y 5.77,Z 553.45,A -85,B 0,C 180,E1 -31229.996,E2 -31229.996} C_VEL
LIN {X 0,Y 14.872,Z 552.813,A -85,B 0,C 180,E1 -31300.927,E2 -31300.927} C_VEL
LIN {X 0,Y 28.306,Z 550.84,A -85,B 0,C 180,E1 -31313.271,E2 -31313.271} C_VEL
LIN {X 0,Y 42.205,Z 547.483,A -85,B 0,C 180,E1 -31317.57,E2 -31317.57} C_VEL
LIN {X 0,Y 49.203,Z 545.257,A -85,B 0,C 180,E1 -31318.913,E2 -31318.913} C_VEL
LIN {X 0,Y 50.828,Z 544.689,A -85,B 0,C 180,E1 -31319.999,E2 -31319.999} C_VEL
LIN {X 0,Y 42.184,Z 547.511,A -85,B 0,C 180,E1 -31321.665,E2 -31321.665} C_VEL
LIN {X 0,Y 28.26,Z 550.898,A -85,B 0,C 180,E1 -31325.891,E2 -31325.891} C_VEL
LIN {X 0,Y 14.773,Z 552.9,A -85,B 0,C 180,E1 -31337.938,E2 -31337.938} C_VEL
LIN {X 0,Y 8.765,Z 553.396,A -85,B 0,C 180,E1 -31356.703,E2 -31356.703} C_VEL
LIN {X 0,Y 5.688,Z 553.557,A -85,B 0,C 180,E1 -31410.004,E2 -31410.004} C_VEL
LIN {X 0,Y 8.766,Z 553.378,A -85,B 0,C 180,E1 -31463.296,E2 -31463.296} C_VEL
LIN {X 0,Y 21.411,Z 552.018,A -85,B 0,C 180,E1 -31489.967,E2 -31489.967} C_VEL
LIN {X 0,Y 35.202,Z 549.301,A -85,B 0,C 180,E1 -31496.584,E2 -31496.584} C_VEL
LIN {X 0,Y 49.196,Z 545.147,A -85,B 0,C 180,E1 -31499.817,E2 -31499.817} C_VEL
LIN {X 0,Y 50.341,Z 544.74,A -85,B 0,C 180,E1 -31500.001,E2 -31500.001} C_VEL
LIN {X 0,Y 49.205,Z 545.136,A -85,B 0,C 180,E1 -31501.13,E2 -31501.13} C_VEL
LIN {X 0,Y 40.617,Z 547.809,A -85,B 0,C 180,E1 -31502.867,E2 -31502.867} C_VEL
LIN {X 0,Y 39.15,Z 549.742,A -85,B 0,C 180,E1 -31503.22,E2 -31503.22} C_VEL
LIN {X 0,Y 39.15,Z 600,A -85,B 0,C 180,E1 -31503.22,E2 -31503.22} C_VEL
LIN {X 0,Y 39.15,Z 600,A -85,B 0,C 180,E1 -31503.22,E2 -31503.22}

QRS_NEXT_CUT()

QRS_NEXT()
QRS_HOME()

END
